(* Logix 5000 project; controller reports 1756-L63 rev 20.11; software revision 20.04; part 23 of 52 *)

        [1504].log_data[0].minminute := 40, [1504].log_data[0].maxminute := 40, [1504].log_data[0].valid := 1, [1504].log_data[1].valid := 1, [1504].log_data[2].valid := 1, [1504].log_data[3].valid := 1, [1504].log_data[4].valid := 1, [1504].log_data[5].valid := 1, [1504].log_data[6].valid := 1, [1504].log_data[7].valid := 1, [1504].log_data[8].valid := 1, [1504].log_data[9].valid := 1, [1504].log_data[10].valid := 1, [1504].log_data[11].valid := 1, [1504].log_data[12].valid := 1, [1504].log_data[13].valid := 1, [1504].log_data[14].valid := 1, [1504].log_data[15].valid := 1, [1504].log_data[16].valid := 1, [1504].log_data[17].valid := 1, [1504].log_data[18].valid := 1, [1504].log_data[19].valid := 1, [1504].time.Year := 2023, [1504].time.Month := 1, [1504].time.Day := 14, [1504].time.Hour := 21, [1504].time.Minute := 44, [1504].time.Second := 59, [1505].log_data[0].min := 1.0, [1505].log_data[0].max := 1.0, [1505].log_data[0].total := 300.0, [1505].log_data[0].time := 300.0, [1505].log_data[0].minminute := 45, [1505].log_data[0].maxminute := 45, [1505].log_data[0].valid := 1, [1505].log_data[1].valid := 1, [1505].log_data[2].valid := 1, [1505].log_data[3].valid := 1, [1505].log_data[4].valid := 1, [1505].log_data[5].valid := 1, [1505].log_data[6].valid := 1, [1505].log_data[7].valid := 1, [1505].log_data[8].valid := 1, [1505].log_data[9].valid := 1, [1505].log_data[10].valid := 1, [1505].log_data[11].valid := 1, [1505].log_data[12].valid := 1, [1505].log_data[13].valid := 1, [1505].log_data[14].valid := 1, [1505].log_data[15].valid := 1, [1505].log_data[16].valid := 1, [1505].log_data[17].valid := 1, [1505].log_data[18].valid := 1, [1505].log_data[19].valid := 1, [1505].time.Year := 2023, [1505].time.Month := 1, [1505].time.Day := 14, [1505].time.Hour := 21, [1505].time.Minute := 49, [1505].time.Second := 59,
        [1506].log_data[0].min := 1.0, [1506].log_data[0].max := 1.0, [1506].log_data[0].total := 300.0, [1506].log_data[0].time := 300.0, [1506].log_data[0].minminute := 50, [1506].log_data[0].maxminute := 50, [1506].log_data[0].valid := 1, [1506].log_data[1].valid := 1, [1506].log_data[2].valid := 1, [1506].log_data[3].valid := 1, [1506].log_data[4].valid := 1, [1506].log_data[5].valid := 1, [1506].log_data[6].valid := 1, [1506].log_data[7].valid := 1, [1506].log_data[8].valid := 1, [1506].log_data[9].valid := 1, [1506].log_data[10].valid := 1, [1506].log_data[11].valid := 1, [1506].log_data[12].valid := 1, [1506].log_data[13].valid := 1, [1506].log_data[14].valid := 1, [1506].log_data[15].valid := 1, [1506].log_data[16].valid := 1, [1506].log_data[17].valid := 1, [1506].log_data[18].valid := 1, [1506].log_data[19].valid := 1, [1506].time.Year := 2023, [1506].time.Month := 1, [1506].time.Day := 14, [1506].time.Hour := 21, [1506].time.Minute := 54, [1506].time.Second := 59, [1507].log_data[0].min := 1.0, [1507].log_data[0].max := 1.0, [1507].log_data[0].total := 300.0, [1507].log_data[0].time := 300.0, [1507].log_data[0].minminute := 55, [1507].log_data[0].maxminute := 55, [1507].log_data[0].valid := 1, [1507].log_data[1].valid := 1, [1507].log_data[2].valid := 1, [1507].log_data[3].valid := 1, [1507].log_data[4].valid := 1, [1507].log_data[5].valid := 1, [1507].log_data[6].valid := 1, [1507].log_data[7].valid := 1, [1507].log_data[8].valid := 1, [1507].log_data[9].valid := 1, [1507].log_data[10].valid := 1, [1507].log_data[11].valid := 1, [1507].log_data[12].valid := 1, [1507].log_data[13].valid := 1, [1507].log_data[14].valid := 1, [1507].log_data[15].valid := 1, [1507].log_data[16].valid := 1, [1507].log_data[17].valid := 1, [1507].log_data[18].valid := 1, [1507].log_data[19].valid := 1, [1507].time.Year := 2023, [1507].time.Month := 1,
        [1507].time.Day := 14, [1507].time.Hour := 21, [1507].time.Minute := 59, [1507].time.Second := 59, [1508].log_data[0].min := 1.0, [1508].log_data[0].max := 1.0, [1508].log_data[0].total := 300.0, [1508].log_data[0].time := 300.0, [1508].log_data[0].valid := 1, [1508].log_data[1].valid := 1, [1508].log_data[2].valid := 1, [1508].log_data[3].valid := 1, [1508].log_data[4].valid := 1, [1508].log_data[5].valid := 1, [1508].log_data[6].valid := 1, [1508].log_data[7].valid := 1, [1508].log_data[8].valid := 1, [1508].log_data[9].valid := 1, [1508].log_data[10].valid := 1, [1508].log_data[11].valid := 1, [1508].log_data[12].valid := 1, [1508].log_data[13].valid := 1, [1508].log_data[14].valid := 1, [1508].log_data[15].valid := 1, [1508].log_data[16].valid := 1, [1508].log_data[17].valid := 1, [1508].log_data[18].valid := 1, [1508].log_data[19].valid := 1, [1508].time.Year := 2023, [1508].time.Month := 1, [1508].time.Day := 14, [1508].time.Hour := 22, [1508].time.Minute := 4, [1508].time.Second := 59, [1509].log_data[0].min := 1.0, [1509].log_data[0].max := 1.0, [1509].log_data[0].total := 300.0, [1509].log_data[0].time := 300.0, [1509].log_data[0].minminute := 5, [1509].log_data[0].maxminute := 5, [1509].log_data[0].valid := 1, [1509].log_data[1].valid := 1, [1509].log_data[2].valid := 1, [1509].log_data[3].valid := 1, [1509].log_data[4].valid := 1, [1509].log_data[5].valid := 1, [1509].log_data[6].valid := 1, [1509].log_data[7].valid := 1, [1509].log_data[8].valid := 1, [1509].log_data[9].valid := 1, [1509].log_data[10].valid := 1, [1509].log_data[11].valid := 1, [1509].log_data[12].valid := 1, [1509].log_data[13].valid := 1, [1509].log_data[14].valid := 1, [1509].log_data[15].valid := 1, [1509].log_data[16].valid := 1, [1509].log_data[17].valid := 1, [1509].log_data[18].valid := 1, [1509].log_data[19].valid := 1,
        [1509].time.Year := 2023, [1509].time.Month := 1, [1509].time.Day := 14, [1509].time.Hour := 22, [1509].time.Minute := 9, [1509].time.Second := 59, [1510].log_data[0].min := 1.0, [1510].log_data[0].max := 1.0, [1510].log_data[0].total := 300.0, [1510].log_data[0].time := 300.0, [1510].log_data[0].minminute := 10, [1510].log_data[0].maxminute := 10, [1510].log_data[0].valid := 1, [1510].log_data[1].valid := 1, [1510].log_data[2].valid := 1, [1510].log_data[3].valid := 1, [1510].log_data[4].valid := 1, [1510].log_data[5].valid := 1, [1510].log_data[6].valid := 1, [1510].log_data[7].valid := 1, [1510].log_data[8].valid := 1, [1510].log_data[9].valid := 1, [1510].log_data[10].valid := 1, [1510].log_data[11].valid := 1, [1510].log_data[12].valid := 1, [1510].log_data[13].valid := 1, [1510].log_data[14].valid := 1, [1510].log_data[15].valid := 1, [1510].log_data[16].valid := 1, [1510].log_data[17].valid := 1, [1510].log_data[18].valid := 1, [1510].log_data[19].valid := 1, [1510].time.Year := 2023, [1510].time.Month := 1, [1510].time.Day := 14, [1510].time.Hour := 22, [1510].time.Minute := 14, [1510].time.Second := 59, [1511].log_data[0].min := 1.0, [1511].log_data[0].max := 1.0, [1511].log_data[0].total := 300.0, [1511].log_data[0].time := 300.0, [1511].log_data[0].minminute := 15, [1511].log_data[0].maxminute := 15, [1511].log_data[0].valid := 1, [1511].log_data[1].valid := 1, [1511].log_data[2].valid := 1, [1511].log_data[3].valid := 1, [1511].log_data[4].valid := 1, [1511].log_data[5].valid := 1, [1511].log_data[6].valid := 1, [1511].log_data[7].valid := 1, [1511].log_data[8].valid := 1, [1511].log_data[9].valid := 1, [1511].log_data[10].valid := 1, [1511].log_data[11].valid := 1, [1511].log_data[12].valid := 1, [1511].log_data[13].valid := 1, [1511].log_data[14].valid := 1, [1511].log_data[15].valid := 1,
        [1511].log_data[16].valid := 1, [1511].log_data[17].valid := 1, [1511].log_data[18].valid := 1, [1511].log_data[19].valid := 1, [1511].time.Year := 2023, [1511].time.Month := 1, [1511].time.Day := 14, [1511].time.Hour := 22, [1511].time.Minute := 19, [1511].time.Second := 59, [1512].log_data[0].min := 1.0, [1512].log_data[0].max := 1.0, [1512].log_data[0].total := 300.0, [1512].log_data[0].time := 300.0, [1512].log_data[0].minminute := 20, [1512].log_data[0].maxminute := 20, [1512].log_data[0].valid := 1, [1512].log_data[1].valid := 1, [1512].log_data[2].valid := 1, [1512].log_data[3].valid := 1, [1512].log_data[4].valid := 1, [1512].log_data[5].valid := 1, [1512].log_data[6].valid := 1, [1512].log_data[7].valid := 1, [1512].log_data[8].valid := 1, [1512].log_data[9].valid := 1, [1512].log_data[10].valid := 1, [1512].log_data[11].valid := 1, [1512].log_data[12].valid := 1, [1512].log_data[13].valid := 1, [1512].log_data[14].valid := 1, [1512].log_data[15].valid := 1, [1512].log_data[16].valid := 1, [1512].log_data[17].valid := 1, [1512].log_data[18].valid := 1, [1512].log_data[19].valid := 1, [1512].time.Year := 2023, [1512].time.Month := 1, [1512].time.Day := 14, [1512].time.Hour := 22, [1512].time.Minute := 24, [1512].time.Second := 59, [1513].log_data[0].min := 1.0, [1513].log_data[0].max := 1.0, [1513].log_data[0].total := 300.0, [1513].log_data[0].time := 300.0, [1513].log_data[0].minminute := 25, [1513].log_data[0].maxminute := 25, [1513].log_data[0].valid := 1, [1513].log_data[1].valid := 1, [1513].log_data[2].valid := 1, [1513].log_data[3].valid := 1, [1513].log_data[4].valid := 1, [1513].log_data[5].valid := 1, [1513].log_data[6].valid := 1, [1513].log_data[7].valid := 1, [1513].log_data[8].valid := 1, [1513].log_data[9].valid := 1, [1513].log_data[10].valid := 1, [1513].log_data[11].valid := 1,
        [1513].log_data[12].valid := 1, [1513].log_data[13].valid := 1, [1513].log_data[14].valid := 1, [1513].log_data[15].valid := 1, [1513].log_data[16].valid := 1, [1513].log_data[17].valid := 1, [1513].log_data[18].valid := 1, [1513].log_data[19].valid := 1, [1513].time.Year := 2023, [1513].time.Month := 1, [1513].time.Day := 14, [1513].time.Hour := 22, [1513].time.Minute := 29, [1513].time.Second := 59, [1514].log_data[0].min := 1.0, [1514].log_data[0].max := 1.0, [1514].log_data[0].total := 300.0, [1514].log_data[0].time := 300.0, [1514].log_data[0].minminute := 30, [1514].log_data[0].maxminute := 30, [1514].log_data[0].valid := 1, [1514].log_data[1].valid := 1, [1514].log_data[2].valid := 1, [1514].log_data[3].valid := 1, [1514].log_data[4].valid := 1, [1514].log_data[5].valid := 1, [1514].log_data[6].valid := 1, [1514].log_data[7].valid := 1, [1514].log_data[8].valid := 1, [1514].log_data[9].valid := 1, [1514].log_data[10].valid := 1, [1514].log_data[11].valid := 1, [1514].log_data[12].valid := 1, [1514].log_data[13].valid := 1, [1514].log_data[14].valid := 1, [1514].log_data[15].valid := 1, [1514].log_data[16].valid := 1, [1514].log_data[17].valid := 1, [1514].log_data[18].valid := 1, [1514].log_data[19].valid := 1, [1514].time.Year := 2023, [1514].time.Month := 1, [1514].time.Day := 14, [1514].time.Hour := 22, [1514].time.Minute := 34, [1514].time.Second := 59, [1515].log_data[0].min := 1.0, [1515].log_data[0].max := 1.0, [1515].log_data[0].total := 300.0, [1515].log_data[0].time := 300.0, [1515].log_data[0].minminute := 35, [1515].log_data[0].maxminute := 35, [1515].log_data[0].valid := 1, [1515].log_data[1].valid := 1, [1515].log_data[2].valid := 1, [1515].log_data[3].valid := 1, [1515].log_data[4].valid := 1, [1515].log_data[5].valid := 1, [1515].log_data[6].valid := 1, [1515].log_data[7].valid := 1,
        [1515].log_data[8].valid := 1, [1515].log_data[9].valid := 1, [1515].log_data[10].valid := 1, [1515].log_data[11].valid := 1, [1515].log_data[12].valid := 1, [1515].log_data[13].valid := 1, [1515].log_data[14].valid := 1, [1515].log_data[15].valid := 1, [1515].log_data[16].valid := 1, [1515].log_data[17].valid := 1, [1515].log_data[18].valid := 1, [1515].log_data[19].valid := 1, [1515].time.Year := 2023, [1515].time.Month := 1, [1515].time.Day := 14, [1515].time.Hour := 22, [1515].time.Minute := 39, [1515].time.Second := 59, [1516].log_data[0].min := 1.0, [1516].log_data[0].max := 1.0, [1516].log_data[0].total := 300.0, [1516].log_data[0].time := 300.0, [1516].log_data[0].minminute := 40, [1516].log_data[0].maxminute := 40, [1516].log_data[0].valid := 1, [1516].log_data[1].valid := 1, [1516].log_data[2].valid := 1, [1516].log_data[3].valid := 1, [1516].log_data[4].valid := 1, [1516].log_data[5].valid := 1, [1516].log_data[6].valid := 1, [1516].log_data[7].valid := 1, [1516].log_data[8].valid := 1, [1516].log_data[9].valid := 1, [1516].log_data[10].valid := 1, [1516].log_data[11].valid := 1, [1516].log_data[12].valid := 1, [1516].log_data[13].valid := 1, [1516].log_data[14].valid := 1, [1516].log_data[15].valid := 1, [1516].log_data[16].valid := 1, [1516].log_data[17].valid := 1, [1516].log_data[18].valid := 1, [1516].log_data[19].valid := 1, [1516].time.Year := 2023, [1516].time.Month := 1, [1516].time.Day := 14, [1516].time.Hour := 22, [1516].time.Minute := 44, [1516].time.Second := 59, [1517].log_data[0].min := 1.0, [1517].log_data[0].max := 1.0, [1517].log_data[0].total := 300.0, [1517].log_data[0].time := 300.0, [1517].log_data[0].minminute := 45, [1517].log_data[0].maxminute := 45, [1517].log_data[0].valid := 1, [1517].log_data[1].valid := 1, [1517].log_data[2].valid := 1, [1517].log_data[3].valid := 1,
        [1517].log_data[4].valid := 1, [1517].log_data[5].valid := 1, [1517].log_data[6].valid := 1, [1517].log_data[7].valid := 1, [1517].log_data[8].valid := 1, [1517].log_data[9].valid := 1, [1517].log_data[10].valid := 1, [1517].log_data[11].valid := 1, [1517].log_data[12].valid := 1, [1517].log_data[13].valid := 1, [1517].log_data[14].valid := 1, [1517].log_data[15].valid := 1, [1517].log_data[16].valid := 1, [1517].log_data[17].valid := 1, [1517].log_data[18].valid := 1, [1517].log_data[19].valid := 1, [1517].time.Year := 2023, [1517].time.Month := 1, [1517].time.Day := 14, [1517].time.Hour := 22, [1517].time.Minute := 49, [1517].time.Second := 59, [1518].log_data[0].min := 1.0, [1518].log_data[0].max := 1.0, [1518].log_data[0].total := 300.0, [1518].log_data[0].time := 300.0, [1518].log_data[0].minminute := 50, [1518].log_data[0].maxminute := 50, [1518].log_data[0].valid := 1, [1518].log_data[1].valid := 1, [1518].log_data[2].valid := 1, [1518].log_data[3].valid := 1, [1518].log_data[4].valid := 1, [1518].log_data[5].valid := 1, [1518].log_data[6].valid := 1, [1518].log_data[7].valid := 1, [1518].log_data[8].valid := 1, [1518].log_data[9].valid := 1, [1518].log_data[10].valid := 1, [1518].log_data[11].valid := 1, [1518].log_data[12].valid := 1, [1518].log_data[13].valid := 1, [1518].log_data[14].valid := 1, [1518].log_data[15].valid := 1, [1518].log_data[16].valid := 1, [1518].log_data[17].valid := 1, [1518].log_data[18].valid := 1, [1518].log_data[19].valid := 1, [1518].time.Year := 2023, [1518].time.Month := 1, [1518].time.Day := 14, [1518].time.Hour := 22, [1518].time.Minute := 54, [1518].time.Second := 59, [1519].log_data[0].min := 1.0, [1519].log_data[0].max := 1.0, [1519].log_data[0].total := 300.0, [1519].log_data[0].time := 300.0, [1519].log_data[0].minminute := 55, [1519].log_data[0].maxminute := 55,
        [1519].log_data[0].valid := 1, [1519].log_data[1].valid := 1, [1519].log_data[2].valid := 1, [1519].log_data[3].valid := 1, [1519].log_data[4].valid := 1, [1519].log_data[5].valid := 1, [1519].log_data[6].valid := 1, [1519].log_data[7].valid := 1, [1519].log_data[8].valid := 1, [1519].log_data[9].valid := 1, [1519].log_data[10].valid := 1, [1519].log_data[11].valid := 1, [1519].log_data[12].valid := 1, [1519].log_data[13].valid := 1, [1519].log_data[14].valid := 1, [1519].log_data[15].valid := 1, [1519].log_data[16].valid := 1, [1519].log_data[17].valid := 1, [1519].log_data[18].valid := 1, [1519].log_data[19].valid := 1, [1519].time.Year := 2023, [1519].time.Month := 1, [1519].time.Day := 14, [1519].time.Hour := 22, [1519].time.Minute := 59, [1519].time.Second := 59, [1520].log_data[0].min := 1.0, [1520].log_data[0].max := 1.0, [1520].log_data[0].total := 299.5, [1520].log_data[0].time := 299.5, [1520].log_data[0].valid := 1, [1520].log_data[1].valid := 1, [1520].log_data[2].valid := 1, [1520].log_data[3].valid := 1, [1520].log_data[4].valid := 1, [1520].log_data[5].valid := 1, [1520].log_data[6].valid := 1, [1520].log_data[7].valid := 1, [1520].log_data[8].valid := 1, [1520].log_data[9].valid := 1, [1520].log_data[10].valid := 1, [1520].log_data[11].valid := 1, [1520].log_data[12].valid := 1, [1520].log_data[13].valid := 1, [1520].log_data[14].valid := 1, [1520].log_data[15].valid := 1, [1520].log_data[16].valid := 1, [1520].log_data[17].valid := 1, [1520].log_data[18].valid := 1, [1520].log_data[19].valid := 1, [1520].time.Year := 2023, [1520].time.Month := 1, [1520].time.Day := 14, [1520].time.Hour := 23, [1520].time.Minute := 4, [1520].time.Second := 59, [1521].log_data[0].min := 1.0, [1521].log_data[0].max := 1.0, [1521].log_data[0].total := 300.0, [1521].log_data[0].time := 300.0,
        [1521].log_data[0].minminute := 5, [1521].log_data[0].maxminute := 5, [1521].log_data[0].valid := 1, [1521].log_data[1].valid := 1, [1521].log_data[2].valid := 1, [1521].log_data[3].valid := 1, [1521].log_data[4].valid := 1, [1521].log_data[5].valid := 1, [1521].log_data[6].valid := 1, [1521].log_data[7].valid := 1, [1521].log_data[8].valid := 1, [1521].log_data[9].valid := 1, [1521].log_data[10].valid := 1, [1521].log_data[11].valid := 1, [1521].log_data[12].valid := 1, [1521].log_data[13].valid := 1, [1521].log_data[14].valid := 1, [1521].log_data[15].valid := 1, [1521].log_data[16].valid := 1, [1521].log_data[17].valid := 1, [1521].log_data[18].valid := 1, [1521].log_data[19].valid := 1, [1521].time.Year := 2023, [1521].time.Month := 1, [1521].time.Day := 14, [1521].time.Hour := 23, [1521].time.Minute := 9, [1521].time.Second := 59, [1522].log_data[0].min := 1.0, [1522].log_data[0].max := 1.0, [1522].log_data[0].total := 300.0, [1522].log_data[0].time := 300.0, [1522].log_data[0].minminute := 10, [1522].log_data[0].maxminute := 10, [1522].log_data[0].valid := 1, [1522].log_data[1].valid := 1, [1522].log_data[2].valid := 1, [1522].log_data[3].valid := 1, [1522].log_data[4].valid := 1, [1522].log_data[5].valid := 1, [1522].log_data[6].valid := 1, [1522].log_data[7].valid := 1, [1522].log_data[8].valid := 1, [1522].log_data[9].valid := 1, [1522].log_data[10].valid := 1, [1522].log_data[11].valid := 1, [1522].log_data[12].valid := 1, [1522].log_data[13].valid := 1, [1522].log_data[14].valid := 1, [1522].log_data[15].valid := 1, [1522].log_data[16].valid := 1, [1522].log_data[17].valid := 1, [1522].log_data[18].valid := 1, [1522].log_data[19].valid := 1, [1522].time.Year := 2023, [1522].time.Month := 1, [1522].time.Day := 14, [1522].time.Hour := 23, [1522].time.Minute := 14, [1522].time.Second := 59,
        [1523].log_data[0].min := 1.0, [1523].log_data[0].max := 1.0, [1523].log_data[0].total := 300.0, [1523].log_data[0].time := 300.0, [1523].log_data[0].minminute := 15, [1523].log_data[0].maxminute := 15, [1523].log_data[0].valid := 1, [1523].log_data[1].valid := 1, [1523].log_data[2].valid := 1, [1523].log_data[3].valid := 1, [1523].log_data[4].valid := 1, [1523].log_data[5].valid := 1, [1523].log_data[6].valid := 1, [1523].log_data[7].valid := 1, [1523].log_data[8].valid := 1, [1523].log_data[9].valid := 1, [1523].log_data[10].valid := 1, [1523].log_data[11].valid := 1, [1523].log_data[12].valid := 1, [1523].log_data[13].valid := 1, [1523].log_data[14].valid := 1, [1523].log_data[15].valid := 1, [1523].log_data[16].valid := 1, [1523].log_data[17].valid := 1, [1523].log_data[18].valid := 1, [1523].log_data[19].valid := 1, [1523].time.Year := 2023, [1523].time.Month := 1, [1523].time.Day := 14, [1523].time.Hour := 23, [1523].time.Minute := 19, [1523].time.Second := 59, [1524].log_data[0].min := 1.0, [1524].log_data[0].max := 1.0, [1524].log_data[0].total := 300.0, [1524].log_data[0].time := 300.0, [1524].log_data[0].minminute := 20, [1524].log_data[0].maxminute := 20, [1524].log_data[0].valid := 1, [1524].log_data[1].valid := 1, [1524].log_data[2].valid := 1, [1524].log_data[3].valid := 1, [1524].log_data[4].valid := 1, [1524].log_data[5].valid := 1, [1524].log_data[6].valid := 1, [1524].log_data[7].valid := 1, [1524].log_data[8].valid := 1, [1524].log_data[9].valid := 1, [1524].log_data[10].valid := 1, [1524].log_data[11].valid := 1, [1524].log_data[12].valid := 1, [1524].log_data[13].valid := 1, [1524].log_data[14].valid := 1, [1524].log_data[15].valid := 1, [1524].log_data[16].valid := 1, [1524].log_data[17].valid := 1, [1524].log_data[18].valid := 1, [1524].log_data[19].valid := 1, [1524].time.Year := 2023, [1524].time.Month := 1,
        [1524].time.Day := 14, [1524].time.Hour := 23, [1524].time.Minute := 24, [1524].time.Second := 59, [1525].log_data[0].min := 1.0, [1525].log_data[0].max := 1.0, [1525].log_data[0].total := 300.0, [1525].log_data[0].time := 300.0, [1525].log_data[0].minminute := 25, [1525].log_data[0].maxminute := 25, [1525].log_data[0].valid := 1, [1525].log_data[1].valid := 1, [1525].log_data[2].valid := 1, [1525].log_data[3].valid := 1, [1525].log_data[4].valid := 1, [1525].log_data[5].valid := 1, [1525].log_data[6].valid := 1, [1525].log_data[7].valid := 1, [1525].log_data[8].valid := 1, [1525].log_data[9].valid := 1, [1525].log_data[10].valid := 1, [1525].log_data[11].valid := 1, [1525].log_data[12].valid := 1, [1525].log_data[13].valid := 1, [1525].log_data[14].valid := 1, [1525].log_data[15].valid := 1, [1525].log_data[16].valid := 1, [1525].log_data[17].valid := 1, [1525].log_data[18].valid := 1, [1525].log_data[19].valid := 1, [1525].time.Year := 2023, [1525].time.Month := 1, [1525].time.Day := 14, [1525].time.Hour := 23, [1525].time.Minute := 29, [1525].time.Second := 59, [1526].log_data[0].min := 1.0, [1526].log_data[0].max := 1.0, [1526].log_data[0].total := 300.0, [1526].log_data[0].time := 300.0, [1526].log_data[0].minminute := 30, [1526].log_data[0].maxminute := 30, [1526].log_data[0].valid := 1, [1526].log_data[1].valid := 1, [1526].log_data[2].valid := 1, [1526].log_data[3].valid := 1, [1526].log_data[4].valid := 1, [1526].log_data[5].valid := 1, [1526].log_data[6].valid := 1, [1526].log_data[7].valid := 1, [1526].log_data[8].valid := 1, [1526].log_data[9].valid := 1, [1526].log_data[10].valid := 1, [1526].log_data[11].valid := 1, [1526].log_data[12].valid := 1, [1526].log_data[13].valid := 1, [1526].log_data[14].valid := 1, [1526].log_data[15].valid := 1, [1526].log_data[16].valid := 1, [1526].log_data[17].valid := 1,
        [1526].log_data[18].valid := 1, [1526].log_data[19].valid := 1, [1526].time.Year := 2023, [1526].time.Month := 1, [1526].time.Day := 14, [1526].time.Hour := 23, [1526].time.Minute := 34, [1526].time.Second := 59, [1527].log_data[0].min := 1.0, [1527].log_data[0].max := 1.0, [1527].log_data[0].total := 300.0, [1527].log_data[0].time := 300.0, [1527].log_data[0].minminute := 35, [1527].log_data[0].maxminute := 35, [1527].log_data[0].valid := 1, [1527].log_data[1].valid := 1, [1527].log_data[2].valid := 1, [1527].log_data[3].valid := 1, [1527].log_data[4].valid := 1, [1527].log_data[5].valid := 1, [1527].log_data[6].valid := 1, [1527].log_data[7].valid := 1, [1527].log_data[8].valid := 1, [1527].log_data[9].valid := 1, [1527].log_data[10].valid := 1, [1527].log_data[11].valid := 1, [1527].log_data[12].valid := 1, [1527].log_data[13].valid := 1, [1527].log_data[14].valid := 1, [1527].log_data[15].valid := 1, [1527].log_data[16].valid := 1, [1527].log_data[17].valid := 1, [1527].log_data[18].valid := 1, [1527].log_data[19].valid := 1, [1527].time.Year := 2023, [1527].time.Month := 1, [1527].time.Day := 14, [1527].time.Hour := 23, [1527].time.Minute := 39, [1527].time.Second := 59, [1528].log_data[0].min := 1.0, [1528].log_data[0].max := 1.0, [1528].log_data[0].total := 300.0, [1528].log_data[0].time := 300.0, [1528].log_data[0].minminute := 40, [1528].log_data[0].maxminute := 40, [1528].log_data[0].valid := 1, [1528].log_data[1].valid := 1, [1528].log_data[2].valid := 1, [1528].log_data[3].valid := 1, [1528].log_data[4].valid := 1, [1528].log_data[5].valid := 1, [1528].log_data[6].valid := 1, [1528].log_data[7].valid := 1, [1528].log_data[8].valid := 1, [1528].log_data[9].valid := 1, [1528].log_data[10].valid := 1, [1528].log_data[11].valid := 1, [1528].log_data[12].valid := 1, [1528].log_data[13].valid := 1,
        [1528].log_data[14].valid := 1, [1528].log_data[15].valid := 1, [1528].log_data[16].valid := 1, [1528].log_data[17].valid := 1, [1528].log_data[18].valid := 1, [1528].log_data[19].valid := 1, [1528].time.Year := 2023, [1528].time.Month := 1, [1528].time.Day := 14, [1528].time.Hour := 23, [1528].time.Minute := 44, [1528].time.Second := 59, [1529].log_data[0].min := 1.0, [1529].log_data[0].max := 1.0, [1529].log_data[0].total := 300.0, [1529].log_data[0].time := 300.0, [1529].log_data[0].minminute := 45, [1529].log_data[0].maxminute := 45, [1529].log_data[0].valid := 1, [1529].log_data[1].valid := 1, [1529].log_data[2].valid := 1, [1529].log_data[3].valid := 1, [1529].log_data[4].valid := 1, [1529].log_data[5].valid := 1, [1529].log_data[6].valid := 1, [1529].log_data[7].valid := 1, [1529].log_data[8].valid := 1, [1529].log_data[9].valid := 1, [1529].log_data[10].valid := 1, [1529].log_data[11].valid := 1, [1529].log_data[12].valid := 1, [1529].log_data[13].valid := 1, [1529].log_data[14].valid := 1, [1529].log_data[15].valid := 1, [1529].log_data[16].valid := 1, [1529].log_data[17].valid := 1, [1529].log_data[18].valid := 1, [1529].log_data[19].valid := 1, [1529].time.Year := 2023, [1529].time.Month := 1, [1529].time.Day := 14, [1529].time.Hour := 23, [1529].time.Minute := 49, [1529].time.Second := 59, [1530].log_data[0].min := 1.0, [1530].log_data[0].max := 1.0, [1530].log_data[0].total := 300.0, [1530].log_data[0].time := 300.0, [1530].log_data[0].minminute := 50, [1530].log_data[0].maxminute := 50, [1530].log_data[0].valid := 1, [1530].log_data[1].valid := 1, [1530].log_data[2].valid := 1, [1530].log_data[3].valid := 1, [1530].log_data[4].valid := 1, [1530].log_data[5].valid := 1, [1530].log_data[6].valid := 1, [1530].log_data[7].valid := 1, [1530].log_data[8].valid := 1, [1530].log_data[9].valid := 1,
        [1530].log_data[10].valid := 1, [1530].log_data[11].valid := 1, [1530].log_data[12].valid := 1, [1530].log_data[13].valid := 1, [1530].log_data[14].valid := 1, [1530].log_data[15].valid := 1, [1530].log_data[16].valid := 1, [1530].log_data[17].valid := 1, [1530].log_data[18].valid := 1, [1530].log_data[19].valid := 1, [1530].time.Year := 2023, [1530].time.Month := 1, [1530].time.Day := 14, [1530].time.Hour := 23, [1530].time.Minute := 54, [1530].time.Second := 59, [1531].log_data[0].min := 1.0, [1531].log_data[0].max := 1.0, [1531].log_data[0].total := 300.0, [1531].log_data[0].time := 300.0, [1531].log_data[0].minminute := 55, [1531].log_data[0].maxminute := 55, [1531].log_data[0].valid := 1, [1531].log_data[1].valid := 1, [1531].log_data[2].valid := 1, [1531].log_data[3].valid := 1, [1531].log_data[4].valid := 1, [1531].log_data[5].valid := 1, [1531].log_data[6].valid := 1, [1531].log_data[7].valid := 1, [1531].log_data[8].valid := 1, [1531].log_data[9].valid := 1, [1531].log_data[10].valid := 1, [1531].log_data[11].valid := 1, [1531].log_data[12].valid := 1, [1531].log_data[13].valid := 1, [1531].log_data[14].valid := 1, [1531].log_data[15].valid := 1, [1531].log_data[16].valid := 1, [1531].log_data[17].valid := 1, [1531].log_data[18].valid := 1, [1531].log_data[19].valid := 1, [1531].time.Year := 2023, [1531].time.Month := 1, [1531].time.Day := 14, [1531].time.Hour := 23, [1531].time.Minute := 59, [1531].time.Second := 59, [1532].log_data[0].min := 1.0, [1532].log_data[0].max := 1.0, [1532].log_data[0].total := 300.0, [1532].log_data[0].time := 300.0, [1532].log_data[0].valid := 1, [1532].log_data[1].valid := 1, [1532].log_data[2].valid := 1, [1532].log_data[3].valid := 1, [1532].log_data[4].valid := 1, [1532].log_data[5].valid := 1, [1532].log_data[6].valid := 1, [1532].log_data[7].valid := 1,
        [1532].log_data[8].valid := 1, [1532].log_data[9].valid := 1, [1532].log_data[10].valid := 1, [1532].log_data[11].valid := 1, [1532].log_data[12].valid := 1, [1532].log_data[13].valid := 1, [1532].log_data[14].valid := 1, [1532].log_data[15].valid := 1, [1532].log_data[16].valid := 1, [1532].log_data[17].valid := 1, [1532].log_data[18].valid := 1, [1532].log_data[19].valid := 1, [1532].time.Year := 2023, [1532].time.Month := 1, [1532].time.Day := 15, [1532].time.Minute := 4, [1532].time.Second := 59, [1533].log_data[0].min := 1.0, [1533].log_data[0].max := 1.0, [1533].log_data[0].total := 300.0, [1533].log_data[0].time := 300.0, [1533].log_data[0].minminute := 5, [1533].log_data[0].maxminute := 5, [1533].log_data[0].valid := 1, [1533].log_data[1].valid := 1, [1533].log_data[2].valid := 1, [1533].log_data[3].valid := 1, [1533].log_data[4].valid := 1, [1533].log_data[5].valid := 1, [1533].log_data[6].valid := 1, [1533].log_data[7].valid := 1, [1533].log_data[8].valid := 1, [1533].log_data[9].valid := 1, [1533].log_data[10].valid := 1, [1533].log_data[11].valid := 1, [1533].log_data[12].valid := 1, [1533].log_data[13].valid := 1, [1533].log_data[14].valid := 1, [1533].log_data[15].valid := 1, [1533].log_data[16].valid := 1, [1533].log_data[17].valid := 1, [1533].log_data[18].valid := 1, [1533].log_data[19].valid := 1, [1533].time.Year := 2023, [1533].time.Month := 1, [1533].time.Day := 15, [1533].time.Minute := 9, [1533].time.Second := 59, [1534].log_data[0].min := 1.0, [1534].log_data[0].max := 1.0, [1534].log_data[0].total := 300.0, [1534].log_data[0].time := 300.0, [1534].log_data[0].minminute := 10, [1534].log_data[0].maxminute := 10, [1534].log_data[0].valid := 1, [1534].log_data[1].valid := 1, [1534].log_data[2].valid := 1, [1534].log_data[3].valid := 1, [1534].log_data[4].valid := 1, [1534].log_data[5].valid := 1,
        [1534].log_data[6].valid := 1, [1534].log_data[7].valid := 1, [1534].log_data[8].valid := 1, [1534].log_data[9].valid := 1, [1534].log_data[10].valid := 1, [1534].log_data[11].valid := 1, [1534].log_data[12].valid := 1, [1534].log_data[13].valid := 1, [1534].log_data[14].valid := 1, [1534].log_data[15].valid := 1, [1534].log_data[16].valid := 1, [1534].log_data[17].valid := 1, [1534].log_data[18].valid := 1, [1534].log_data[19].valid := 1, [1534].time.Year := 2023, [1534].time.Month := 1, [1534].time.Day := 15, [1534].time.Minute := 14, [1534].time.Second := 59, [1535].log_data[0].min := 1.0, [1535].log_data[0].max := 1.0, [1535].log_data[0].total := 300.0, [1535].log_data[0].time := 300.0, [1535].log_data[0].minminute := 15, [1535].log_data[0].maxminute := 15, [1535].log_data[0].valid := 1, [1535].log_data[1].valid := 1, [1535].log_data[2].valid := 1, [1535].log_data[3].valid := 1, [1535].log_data[4].valid := 1, [1535].log_data[5].valid := 1, [1535].log_data[6].valid := 1, [1535].log_data[7].valid := 1, [1535].log_data[8].valid := 1, [1535].log_data[9].valid := 1, [1535].log_data[10].valid := 1, [1535].log_data[11].valid := 1, [1535].log_data[12].valid := 1, [1535].log_data[13].valid := 1, [1535].log_data[14].valid := 1, [1535].log_data[15].valid := 1, [1535].log_data[16].valid := 1, [1535].log_data[17].valid := 1, [1535].log_data[18].valid := 1, [1535].log_data[19].valid := 1, [1535].time.Year := 2023, [1535].time.Month := 1, [1535].time.Day := 15, [1535].time.Minute := 19, [1535].time.Second := 59, [1536].log_data[0].min := 1.0, [1536].log_data[0].max := 1.0, [1536].log_data[0].total := 300.0, [1536].log_data[0].time := 300.0, [1536].log_data[0].minminute := 20, [1536].log_data[0].maxminute := 20, [1536].log_data[0].valid := 1, [1536].log_data[1].valid := 1, [1536].log_data[2].valid := 1, [1536].log_data[3].valid := 1,
        [1536].log_data[4].valid := 1, [1536].log_data[5].valid := 1, [1536].log_data[6].valid := 1, [1536].log_data[7].valid := 1, [1536].log_data[8].valid := 1, [1536].log_data[9].valid := 1, [1536].log_data[10].valid := 1, [1536].log_data[11].valid := 1, [1536].log_data[12].valid := 1, [1536].log_data[13].valid := 1, [1536].log_data[14].valid := 1, [1536].log_data[15].valid := 1, [1536].log_data[16].valid := 1, [1536].log_data[17].valid := 1, [1536].log_data[18].valid := 1, [1536].log_data[19].valid := 1, [1536].time.Year := 2023, [1536].time.Month := 1, [1536].time.Day := 15, [1536].time.Minute := 24, [1536].time.Second := 59, [1537].log_data[0].min := 1.0, [1537].log_data[0].max := 1.0, [1537].log_data[0].total := 300.0, [1537].log_data[0].time := 300.0, [1537].log_data[0].minminute := 25, [1537].log_data[0].maxminute := 25, [1537].log_data[0].valid := 1, [1537].log_data[1].valid := 1, [1537].log_data[2].valid := 1, [1537].log_data[3].valid := 1, [1537].log_data[4].valid := 1, [1537].log_data[5].valid := 1, [1537].log_data[6].valid := 1, [1537].log_data[7].valid := 1, [1537].log_data[8].valid := 1, [1537].log_data[9].valid := 1, [1537].log_data[10].valid := 1, [1537].log_data[11].valid := 1, [1537].log_data[12].valid := 1, [1537].log_data[13].valid := 1, [1537].log_data[14].valid := 1, [1537].log_data[15].valid := 1, [1537].log_data[16].valid := 1, [1537].log_data[17].valid := 1, [1537].log_data[18].valid := 1, [1537].log_data[19].valid := 1, [1537].time.Year := 2023, [1537].time.Month := 1, [1537].time.Day := 15, [1537].time.Minute := 29, [1537].time.Second := 59, [1538].log_data[0].min := 1.0, [1538].log_data[0].max := 1.0, [1538].log_data[0].total := 300.0, [1538].log_data[0].time := 300.0, [1538].log_data[0].minminute := 30, [1538].log_data[0].maxminute := 30, [1538].log_data[0].valid := 1, [1538].log_data[1].valid := 1,
        [1538].log_data[2].valid := 1, [1538].log_data[3].valid := 1, [1538].log_data[4].valid := 1, [1538].log_data[5].valid := 1, [1538].log_data[6].valid := 1, [1538].log_data[7].valid := 1, [1538].log_data[8].valid := 1, [1538].log_data[9].valid := 1, [1538].log_data[10].valid := 1, [1538].log_data[11].valid := 1, [1538].log_data[12].valid := 1, [1538].log_data[13].valid := 1, [1538].log_data[14].valid := 1, [1538].log_data[15].valid := 1, [1538].log_data[16].valid := 1, [1538].log_data[17].valid := 1, [1538].log_data[18].valid := 1, [1538].log_data[19].valid := 1, [1538].time.Year := 2023, [1538].time.Month := 1, [1538].time.Day := 15, [1538].time.Minute := 34, [1538].time.Second := 59, [1539].log_data[0].min := 1.0, [1539].log_data[0].max := 1.0, [1539].log_data[0].total := 300.0, [1539].log_data[0].time := 300.0, [1539].log_data[0].minminute := 35, [1539].log_data[0].maxminute := 35, [1539].log_data[0].valid := 1, [1539].log_data[1].valid := 1, [1539].log_data[2].valid := 1, [1539].log_data[3].valid := 1, [1539].log_data[4].valid := 1, [1539].log_data[5].valid := 1, [1539].log_data[6].valid := 1, [1539].log_data[7].valid := 1, [1539].log_data[8].valid := 1, [1539].log_data[9].valid := 1, [1539].log_data[10].valid := 1, [1539].log_data[11].valid := 1, [1539].log_data[12].valid := 1, [1539].log_data[13].valid := 1, [1539].log_data[14].valid := 1, [1539].log_data[15].valid := 1, [1539].log_data[16].valid := 1, [1539].log_data[17].valid := 1, [1539].log_data[18].valid := 1, [1539].log_data[19].valid := 1, [1539].time.Year := 2023, [1539].time.Month := 1, [1539].time.Day := 15, [1539].time.Minute := 39, [1539].time.Second := 59, [1540].log_data[0].min := 1.0, [1540].log_data[0].max := 1.0, [1540].log_data[0].total := 300.0, [1540].log_data[0].time := 300.0, [1540].log_data[0].minminute := 40, [1540].log_data[0].maxminute := 40,
        [1540].log_data[0].valid := 1, [1540].log_data[1].valid := 1, [1540].log_data[2].valid := 1, [1540].log_data[3].valid := 1, [1540].log_data[4].valid := 1, [1540].log_data[5].valid := 1, [1540].log_data[6].valid := 1, [1540].log_data[7].valid := 1, [1540].log_data[8].valid := 1, [1540].log_data[9].valid := 1, [1540].log_data[10].valid := 1, [1540].log_data[11].valid := 1, [1540].log_data[12].valid := 1, [1540].log_data[13].valid := 1, [1540].log_data[14].valid := 1, [1540].log_data[15].valid := 1, [1540].log_data[16].valid := 1, [1540].log_data[17].valid := 1, [1540].log_data[18].valid := 1, [1540].log_data[19].valid := 1, [1540].time.Year := 2023, [1540].time.Month := 1, [1540].time.Day := 15, [1540].time.Minute := 44, [1540].time.Second := 59, [1541].log_data[0].min := 1.0, [1541].log_data[0].max := 1.0, [1541].log_data[0].total := 300.0, [1541].log_data[0].time := 300.0, [1541].log_data[0].minminute := 45, [1541].log_data[0].maxminute := 45, [1541].log_data[0].valid := 1, [1541].log_data[1].valid := 1, [1541].log_data[2].valid := 1, [1541].log_data[3].valid := 1, [1541].log_data[4].valid := 1, [1541].log_data[5].valid := 1, [1541].log_data[6].valid := 1, [1541].log_data[7].valid := 1, [1541].log_data[8].valid := 1, [1541].log_data[9].valid := 1, [1541].log_data[10].valid := 1, [1541].log_data[11].valid := 1, [1541].log_data[12].valid := 1, [1541].log_data[13].valid := 1, [1541].log_data[14].valid := 1, [1541].log_data[15].valid := 1, [1541].log_data[16].valid := 1, [1541].log_data[17].valid := 1, [1541].log_data[18].valid := 1, [1541].log_data[19].valid := 1, [1541].time.Year := 2023, [1541].time.Month := 1, [1541].time.Day := 15, [1541].time.Minute := 49, [1541].time.Second := 59, [1542].log_data[0].min := 1.0, [1542].log_data[0].max := 1.0, [1542].log_data[0].total := 300.0, [1542].log_data[0].time := 300.0,
        [1542].log_data[0].minminute := 50, [1542].log_data[0].maxminute := 50, [1542].log_data[0].valid := 1, [1542].log_data[1].valid := 1, [1542].log_data[2].valid := 1, [1542].log_data[3].valid := 1, [1542].log_data[4].valid := 1, [1542].log_data[5].valid := 1, [1542].log_data[6].valid := 1, [1542].log_data[7].valid := 1, [1542].log_data[8].valid := 1, [1542].log_data[9].valid := 1, [1542].log_data[10].valid := 1, [1542].log_data[11].valid := 1, [1542].log_data[12].valid := 1, [1542].log_data[13].valid := 1, [1542].log_data[14].valid := 1, [1542].log_data[15].valid := 1, [1542].log_data[16].valid := 1, [1542].log_data[17].valid := 1, [1542].log_data[18].valid := 1, [1542].log_data[19].valid := 1, [1542].time.Year := 2023, [1542].time.Month := 1, [1542].time.Day := 15, [1542].time.Minute := 54, [1542].time.Second := 59, [1543].log_data[0].min := 1.0, [1543].log_data[0].max := 1.0, [1543].log_data[0].total := 300.0, [1543].log_data[0].time := 300.0, [1543].log_data[0].minminute := 55, [1543].log_data[0].maxminute := 55, [1543].log_data[0].valid := 1, [1543].log_data[1].valid := 1, [1543].log_data[2].valid := 1, [1543].log_data[3].valid := 1, [1543].log_data[4].valid := 1, [1543].log_data[5].valid := 1, [1543].log_data[6].valid := 1, [1543].log_data[7].valid := 1, [1543].log_data[8].valid := 1, [1543].log_data[9].valid := 1, [1543].log_data[10].valid := 1, [1543].log_data[11].valid := 1, [1543].log_data[12].valid := 1, [1543].log_data[13].valid := 1, [1543].log_data[14].valid := 1, [1543].log_data[15].valid := 1, [1543].log_data[16].valid := 1, [1543].log_data[17].valid := 1, [1543].log_data[18].valid := 1, [1543].log_data[19].valid := 1, [1543].time.Year := 2023, [1543].time.Month := 1, [1543].time.Day := 15, [1543].time.Minute := 59, [1543].time.Second := 59, [1544].log_data[0].min := 1.0, [1544].log_data[0].max := 1.0,
        [1544].log_data[0].total := 300.0, [1544].log_data[0].time := 300.0, [1544].log_data[0].valid := 1, [1544].log_data[1].valid := 1, [1544].log_data[2].valid := 1, [1544].log_data[3].valid := 1, [1544].log_data[4].valid := 1, [1544].log_data[5].valid := 1, [1544].log_data[6].valid := 1, [1544].log_data[7].valid := 1, [1544].log_data[8].valid := 1, [1544].log_data[9].valid := 1, [1544].log_data[10].valid := 1, [1544].log_data[11].valid := 1, [1544].log_data[12].valid := 1, [1544].log_data[13].valid := 1, [1544].log_data[14].valid := 1, [1544].log_data[15].valid := 1, [1544].log_data[16].valid := 1, [1544].log_data[17].valid := 1, [1544].log_data[18].valid := 1, [1544].log_data[19].valid := 1, [1544].time.Year := 2023, [1544].time.Month := 1, [1544].time.Day := 15, [1544].time.Hour := 1, [1544].time.Minute := 4, [1544].time.Second := 59, [1545].log_data[0].min := 1.0, [1545].log_data[0].max := 1.0, [1545].log_data[0].total := 300.0, [1545].log_data[0].time := 300.0, [1545].log_data[0].minminute := 5, [1545].log_data[0].maxminute := 5, [1545].log_data[0].valid := 1, [1545].log_data[1].valid := 1, [1545].log_data[2].valid := 1, [1545].log_data[3].valid := 1, [1545].log_data[4].valid := 1, [1545].log_data[5].valid := 1, [1545].log_data[6].valid := 1, [1545].log_data[7].valid := 1, [1545].log_data[8].valid := 1, [1545].log_data[9].valid := 1, [1545].log_data[10].valid := 1, [1545].log_data[11].valid := 1, [1545].log_data[12].valid := 1, [1545].log_data[13].valid := 1, [1545].log_data[14].valid := 1, [1545].log_data[15].valid := 1, [1545].log_data[16].valid := 1, [1545].log_data[17].valid := 1, [1545].log_data[18].valid := 1, [1545].log_data[19].valid := 1, [1545].time.Year := 2023, [1545].time.Month := 1, [1545].time.Day := 15, [1545].time.Hour := 1, [1545].time.Minute := 9, [1545].time.Second := 59,
        [1546].log_data[0].min := 1.0, [1546].log_data[0].max := 1.0, [1546].log_data[0].total := 300.0, [1546].log_data[0].time := 300.0, [1546].log_data[0].minminute := 10, [1546].log_data[0].maxminute := 10, [1546].log_data[0].valid := 1, [1546].log_data[1].valid := 1, [1546].log_data[2].valid := 1, [1546].log_data[3].valid := 1, [1546].log_data[4].valid := 1, [1546].log_data[5].valid := 1, [1546].log_data[6].valid := 1, [1546].log_data[7].valid := 1, [1546].log_data[8].valid := 1, [1546].log_data[9].valid := 1, [1546].log_data[10].valid := 1, [1546].log_data[11].valid := 1, [1546].log_data[12].valid := 1, [1546].log_data[13].valid := 1, [1546].log_data[14].valid := 1, [1546].log_data[15].valid := 1, [1546].log_data[16].valid := 1, [1546].log_data[17].valid := 1, [1546].log_data[18].valid := 1, [1546].log_data[19].valid := 1, [1546].time.Year := 2023, [1546].time.Month := 1, [1546].time.Day := 15, [1546].time.Hour := 1, [1546].time.Minute := 14, [1546].time.Second := 59, [1547].log_data[0].min := 1.0, [1547].log_data[0].max := 1.0, [1547].log_data[0].total := 300.0, [1547].log_data[0].time := 300.0, [1547].log_data[0].minminute := 15, [1547].log_data[0].maxminute := 15, [1547].log_data[0].valid := 1, [1547].log_data[1].valid := 1, [1547].log_data[2].valid := 1, [1547].log_data[3].valid := 1, [1547].log_data[4].valid := 1, [1547].log_data[5].valid := 1, [1547].log_data[6].valid := 1, [1547].log_data[7].valid := 1, [1547].log_data[8].valid := 1, [1547].log_data[9].valid := 1, [1547].log_data[10].valid := 1, [1547].log_data[11].valid := 1, [1547].log_data[12].valid := 1, [1547].log_data[13].valid := 1, [1547].log_data[14].valid := 1, [1547].log_data[15].valid := 1, [1547].log_data[16].valid := 1, [1547].log_data[17].valid := 1, [1547].log_data[18].valid := 1, [1547].log_data[19].valid := 1, [1547].time.Year := 2023, [1547].time.Month := 1,
        [1547].time.Day := 15, [1547].time.Hour := 1, [1547].time.Minute := 19, [1547].time.Second := 59, [1548].log_data[0].min := 1.0, [1548].log_data[0].max := 1.0, [1548].log_data[0].total := 300.0, [1548].log_data[0].time := 300.0, [1548].log_data[0].minminute := 20, [1548].log_data[0].maxminute := 20, [1548].log_data[0].valid := 1, [1548].log_data[1].valid := 1, [1548].log_data[2].valid := 1, [1548].log_data[3].valid := 1, [1548].log_data[4].valid := 1, [1548].log_data[5].valid := 1, [1548].log_data[6].valid := 1, [1548].log_data[7].valid := 1, [1548].log_data[8].valid := 1, [1548].log_data[9].valid := 1, [1548].log_data[10].valid := 1, [1548].log_data[11].valid := 1, [1548].log_data[12].valid := 1, [1548].log_data[13].valid := 1, [1548].log_data[14].valid := 1, [1548].log_data[15].valid := 1, [1548].log_data[16].valid := 1, [1548].log_data[17].valid := 1, [1548].log_data[18].valid := 1, [1548].log_data[19].valid := 1, [1548].time.Year := 2023, [1548].time.Month := 1, [1548].time.Day := 15, [1548].time.Hour := 1, [1548].time.Minute := 24, [1548].time.Second := 59, [1549].log_data[0].min := 1.0, [1549].log_data[0].max := 1.0, [1549].log_data[0].total := 300.0, [1549].log_data[0].time := 300.0, [1549].log_data[0].minminute := 25, [1549].log_data[0].maxminute := 25, [1549].log_data[0].valid := 1, [1549].log_data[1].valid := 1, [1549].log_data[2].valid := 1, [1549].log_data[3].valid := 1, [1549].log_data[4].valid := 1, [1549].log_data[5].valid := 1, [1549].log_data[6].valid := 1, [1549].log_data[7].valid := 1, [1549].log_data[8].valid := 1, [1549].log_data[9].valid := 1, [1549].log_data[10].valid := 1, [1549].log_data[11].valid := 1, [1549].log_data[12].valid := 1, [1549].log_data[13].valid := 1, [1549].log_data[14].valid := 1, [1549].log_data[15].valid := 1, [1549].log_data[16].valid := 1, [1549].log_data[17].valid := 1,
        [1549].log_data[18].valid := 1, [1549].log_data[19].valid := 1, [1549].time.Year := 2023, [1549].time.Month := 1, [1549].time.Day := 15, [1549].time.Hour := 1, [1549].time.Minute := 29, [1549].time.Second := 59, [1550].log_data[0].min := 1.0, [1550].log_data[0].max := 1.0, [1550].log_data[0].total := 300.0, [1550].log_data[0].time := 300.0, [1550].log_data[0].minminute := 30, [1550].log_data[0].maxminute := 30, [1550].log_data[0].valid := 1, [1550].log_data[1].valid := 1, [1550].log_data[2].valid := 1, [1550].log_data[3].valid := 1, [1550].log_data[4].valid := 1, [1550].log_data[5].valid := 1, [1550].log_data[6].valid := 1, [1550].log_data[7].valid := 1, [1550].log_data[8].valid := 1, [1550].log_data[9].valid := 1, [1550].log_data[10].valid := 1, [1550].log_data[11].valid := 1, [1550].log_data[12].valid := 1, [1550].log_data[13].valid := 1, [1550].log_data[14].valid := 1, [1550].log_data[15].valid := 1, [1550].log_data[16].valid := 1, [1550].log_data[17].valid := 1, [1550].log_data[18].valid := 1, [1550].log_data[19].valid := 1, [1550].time.Year := 2023, [1550].time.Month := 1, [1550].time.Day := 15, [1550].time.Hour := 1, [1550].time.Minute := 34, [1550].time.Second := 59, [1551].log_data[0].min := 1.0, [1551].log_data[0].max := 1.0, [1551].log_data[0].total := 300.0, [1551].log_data[0].time := 300.0, [1551].log_data[0].minminute := 35, [1551].log_data[0].maxminute := 35, [1551].log_data[0].valid := 1, [1551].log_data[1].valid := 1, [1551].log_data[2].valid := 1, [1551].log_data[3].valid := 1, [1551].log_data[4].valid := 1, [1551].log_data[5].valid := 1, [1551].log_data[6].valid := 1, [1551].log_data[7].valid := 1, [1551].log_data[8].valid := 1, [1551].log_data[9].valid := 1, [1551].log_data[10].valid := 1, [1551].log_data[11].valid := 1, [1551].log_data[12].valid := 1, [1551].log_data[13].valid := 1,
        [1551].log_data[14].valid := 1, [1551].log_data[15].valid := 1, [1551].log_data[16].valid := 1, [1551].log_data[17].valid := 1, [1551].log_data[18].valid := 1, [1551].log_data[19].valid := 1, [1551].time.Year := 2023, [1551].time.Month := 1, [1551].time.Day := 15, [1551].time.Hour := 1, [1551].time.Minute := 39, [1551].time.Second := 59, [1552].log_data[0].min := 1.0, [1552].log_data[0].max := 1.0, [1552].log_data[0].total := 300.0, [1552].log_data[0].time := 300.0, [1552].log_data[0].minminute := 40, [1552].log_data[0].maxminute := 40, [1552].log_data[0].valid := 1, [1552].log_data[1].valid := 1, [1552].log_data[2].valid := 1, [1552].log_data[3].valid := 1, [1552].log_data[4].valid := 1, [1552].log_data[5].valid := 1, [1552].log_data[6].valid := 1, [1552].log_data[7].valid := 1, [1552].log_data[8].valid := 1, [1552].log_data[9].valid := 1, [1552].log_data[10].valid := 1, [1552].log_data[11].valid := 1, [1552].log_data[12].valid := 1, [1552].log_data[13].valid := 1, [1552].log_data[14].valid := 1, [1552].log_data[15].valid := 1, [1552].log_data[16].valid := 1, [1552].log_data[17].valid := 1, [1552].log_data[18].valid := 1, [1552].log_data[19].valid := 1, [1552].time.Year := 2023, [1552].time.Month := 1, [1552].time.Day := 15, [1552].time.Hour := 1, [1552].time.Minute := 44, [1552].time.Second := 59, [1553].log_data[0].min := 1.0, [1553].log_data[0].max := 1.0, [1553].log_data[0].total := 300.0, [1553].log_data[0].time := 300.0, [1553].log_data[0].minminute := 45, [1553].log_data[0].maxminute := 45, [1553].log_data[0].valid := 1, [1553].log_data[1].valid := 1, [1553].log_data[2].valid := 1, [1553].log_data[3].valid := 1, [1553].log_data[4].valid := 1, [1553].log_data[5].valid := 1, [1553].log_data[6].valid := 1, [1553].log_data[7].valid := 1, [1553].log_data[8].valid := 1, [1553].log_data[9].valid := 1,
        [1553].log_data[10].valid := 1, [1553].log_data[11].valid := 1, [1553].log_data[12].valid := 1, [1553].log_data[13].valid := 1, [1553].log_data[14].valid := 1, [1553].log_data[15].valid := 1, [1553].log_data[16].valid := 1, [1553].log_data[17].valid := 1, [1553].log_data[18].valid := 1, [1553].log_data[19].valid := 1, [1553].time.Year := 2023, [1553].time.Month := 1, [1553].time.Day := 15, [1553].time.Hour := 1, [1553].time.Minute := 49, [1553].time.Second := 59, [1554].log_data[0].min := 1.0, [1554].log_data[0].max := 1.0, [1554].log_data[0].total := 300.0, [1554].log_data[0].time := 300.0, [1554].log_data[0].minminute := 50, [1554].log_data[0].maxminute := 50, [1554].log_data[0].valid := 1, [1554].log_data[1].valid := 1, [1554].log_data[2].valid := 1, [1554].log_data[3].valid := 1, [1554].log_data[4].valid := 1, [1554].log_data[5].valid := 1, [1554].log_data[6].valid := 1, [1554].log_data[7].valid := 1, [1554].log_data[8].valid := 1, [1554].log_data[9].valid := 1, [1554].log_data[10].valid := 1, [1554].log_data[11].valid := 1, [1554].log_data[12].valid := 1, [1554].log_data[13].valid := 1, [1554].log_data[14].valid := 1, [1554].log_data[15].valid := 1, [1554].log_data[16].valid := 1, [1554].log_data[17].valid := 1, [1554].log_data[18].valid := 1, [1554].log_data[19].valid := 1, [1554].time.Year := 2023, [1554].time.Month := 1, [1554].time.Day := 15, [1554].time.Hour := 1, [1554].time.Minute := 54, [1554].time.Second := 59, [1555].log_data[0].min := 1.0, [1555].log_data[0].max := 1.0, [1555].log_data[0].total := 300.0, [1555].log_data[0].time := 300.0, [1555].log_data[0].minminute := 55, [1555].log_data[0].maxminute := 55, [1555].log_data[0].valid := 1, [1555].log_data[1].valid := 1, [1555].log_data[2].valid := 1, [1555].log_data[3].valid := 1, [1555].log_data[4].valid := 1, [1555].log_data[5].valid := 1,
        [1555].log_data[6].valid := 1, [1555].log_data[7].valid := 1, [1555].log_data[8].valid := 1, [1555].log_data[9].valid := 1, [1555].log_data[10].valid := 1, [1555].log_data[11].valid := 1, [1555].log_data[12].valid := 1, [1555].log_data[13].valid := 1, [1555].log_data[14].valid := 1, [1555].log_data[15].valid := 1, [1555].log_data[16].valid := 1, [1555].log_data[17].valid := 1, [1555].log_data[18].valid := 1, [1555].log_data[19].valid := 1, [1555].time.Year := 2023, [1555].time.Month := 1, [1555].time.Day := 15, [1555].time.Hour := 1, [1555].time.Minute := 59, [1555].time.Second := 59, [1556].log_data[0].min := 1.0, [1556].log_data[0].max := 1.0, [1556].log_data[0].total := 300.0, [1556].log_data[0].time := 300.0, [1556].log_data[0].valid := 1, [1556].log_data[1].valid := 1, [1556].log_data[2].valid := 1, [1556].log_data[3].valid := 1, [1556].log_data[4].valid := 1, [1556].log_data[5].valid := 1, [1556].log_data[6].valid := 1, [1556].log_data[7].valid := 1, [1556].log_data[8].valid := 1, [1556].log_data[9].valid := 1, [1556].log_data[10].valid := 1, [1556].log_data[11].valid := 1, [1556].log_data[12].valid := 1, [1556].log_data[13].valid := 1, [1556].log_data[14].valid := 1, [1556].log_data[15].valid := 1, [1556].log_data[16].valid := 1, [1556].log_data[17].valid := 1, [1556].log_data[18].valid := 1, [1556].log_data[19].valid := 1, [1556].time.Year := 2023, [1556].time.Month := 1, [1556].time.Day := 15, [1556].time.Hour := 2, [1556].time.Minute := 4, [1556].time.Second := 59, [1557].log_data[0].min := 1.0, [1557].log_data[0].max := 1.0, [1557].log_data[0].total := 300.0, [1557].log_data[0].time := 300.0, [1557].log_data[0].minminute := 5, [1557].log_data[0].maxminute := 5, [1557].log_data[0].valid := 1, [1557].log_data[1].valid := 1, [1557].log_data[2].valid := 1, [1557].log_data[3].valid := 1,
        [1557].log_data[4].valid := 1, [1557].log_data[5].valid := 1, [1557].log_data[6].valid := 1, [1557].log_data[7].valid := 1, [1557].log_data[8].valid := 1, [1557].log_data[9].valid := 1, [1557].log_data[10].valid := 1, [1557].log_data[11].valid := 1, [1557].log_data[12].valid := 1, [1557].log_data[13].valid := 1, [1557].log_data[14].valid := 1, [1557].log_data[15].valid := 1, [1557].log_data[16].valid := 1, [1557].log_data[17].valid := 1, [1557].log_data[18].valid := 1, [1557].log_data[19].valid := 1, [1557].time.Year := 2023, [1557].time.Month := 1, [1557].time.Day := 15, [1557].time.Hour := 2, [1557].time.Minute := 9, [1557].time.Second := 59, [1558].log_data[0].min := 1.0, [1558].log_data[0].max := 1.0, [1558].log_data[0].total := 300.0, [1558].log_data[0].time := 300.0, [1558].log_data[0].minminute := 10, [1558].log_data[0].maxminute := 10, [1558].log_data[0].valid := 1, [1558].log_data[1].valid := 1, [1558].log_data[2].valid := 1, [1558].log_data[3].valid := 1, [1558].log_data[4].valid := 1, [1558].log_data[5].valid := 1, [1558].log_data[6].valid := 1, [1558].log_data[7].valid := 1, [1558].log_data[8].valid := 1, [1558].log_data[9].valid := 1, [1558].log_data[10].valid := 1, [1558].log_data[11].valid := 1, [1558].log_data[12].valid := 1, [1558].log_data[13].valid := 1, [1558].log_data[14].valid := 1, [1558].log_data[15].valid := 1, [1558].log_data[16].valid := 1, [1558].log_data[17].valid := 1, [1558].log_data[18].valid := 1, [1558].log_data[19].valid := 1, [1558].time.Year := 2023, [1558].time.Month := 1, [1558].time.Day := 15, [1558].time.Hour := 2, [1558].time.Minute := 14, [1558].time.Second := 59, [1559].log_data[0].min := 1.0, [1559].log_data[0].max := 1.0, [1559].log_data[0].total := 300.0, [1559].log_data[0].time := 300.0, [1559].log_data[0].minminute := 15, [1559].log_data[0].maxminute := 15,
        [1559].log_data[0].valid := 1, [1559].log_data[1].valid := 1, [1559].log_data[2].valid := 1, [1559].log_data[3].valid := 1, [1559].log_data[4].valid := 1, [1559].log_data[5].valid := 1, [1559].log_data[6].valid := 1, [1559].log_data[7].valid := 1, [1559].log_data[8].valid := 1, [1559].log_data[9].valid := 1, [1559].log_data[10].valid := 1, [1559].log_data[11].valid := 1, [1559].log_data[12].valid := 1, [1559].log_data[13].valid := 1, [1559].log_data[14].valid := 1, [1559].log_data[15].valid := 1, [1559].log_data[16].valid := 1, [1559].log_data[17].valid := 1, [1559].log_data[18].valid := 1, [1559].log_data[19].valid := 1, [1559].time.Year := 2023, [1559].time.Month := 1, [1559].time.Day := 15, [1559].time.Hour := 2, [1559].time.Minute := 19, [1559].time.Second := 59, [1560].log_data[0].min := 1.0, [1560].log_data[0].max := 1.0, [1560].log_data[0].total := 300.0, [1560].log_data[0].time := 300.0, [1560].log_data[0].minminute := 20, [1560].log_data[0].maxminute := 20, [1560].log_data[0].valid := 1, [1560].log_data[1].valid := 1, [1560].log_data[2].valid := 1, [1560].log_data[3].valid := 1, [1560].log_data[4].valid := 1, [1560].log_data[5].valid := 1, [1560].log_data[6].valid := 1, [1560].log_data[7].valid := 1, [1560].log_data[8].valid := 1, [1560].log_data[9].valid := 1, [1560].log_data[10].valid := 1, [1560].log_data[11].valid := 1, [1560].log_data[12].valid := 1, [1560].log_data[13].valid := 1, [1560].log_data[14].valid := 1, [1560].log_data[15].valid := 1, [1560].log_data[16].valid := 1, [1560].log_data[17].valid := 1, [1560].log_data[18].valid := 1, [1560].log_data[19].valid := 1, [1560].time.Year := 2023, [1560].time.Month := 1, [1560].time.Day := 15, [1560].time.Hour := 2, [1560].time.Minute := 24, [1560].time.Second := 59, [1561].log_data[0].min := 1.0, [1561].log_data[0].max := 1.0,
        [1561].log_data[0].total := 300.0, [1561].log_data[0].time := 300.0, [1561].log_data[0].minminute := 25, [1561].log_data[0].maxminute := 25, [1561].log_data[0].valid := 1, [1561].log_data[1].valid := 1, [1561].log_data[2].valid := 1, [1561].log_data[3].valid := 1, [1561].log_data[4].valid := 1, [1561].log_data[5].valid := 1, [1561].log_data[6].valid := 1, [1561].log_data[7].valid := 1, [1561].log_data[8].valid := 1, [1561].log_data[9].valid := 1, [1561].log_data[10].valid := 1, [1561].log_data[11].valid := 1, [1561].log_data[12].valid := 1, [1561].log_data[13].valid := 1, [1561].log_data[14].valid := 1, [1561].log_data[15].valid := 1, [1561].log_data[16].valid := 1, [1561].log_data[17].valid := 1, [1561].log_data[18].valid := 1, [1561].log_data[19].valid := 1, [1561].time.Year := 2023, [1561].time.Month := 1, [1561].time.Day := 15, [1561].time.Hour := 2, [1561].time.Minute := 29, [1561].time.Second := 59, [1562].log_data[0].min := 1.0, [1562].log_data[0].max := 1.0, [1562].log_data[0].total := 300.0, [1562].log_data[0].time := 300.0, [1562].log_data[0].minminute := 30, [1562].log_data[0].maxminute := 30, [1562].log_data[0].valid := 1, [1562].log_data[1].valid := 1, [1562].log_data[2].valid := 1, [1562].log_data[3].valid := 1, [1562].log_data[4].valid := 1, [1562].log_data[5].valid := 1, [1562].log_data[6].valid := 1, [1562].log_data[7].valid := 1, [1562].log_data[8].valid := 1, [1562].log_data[9].valid := 1, [1562].log_data[10].valid := 1, [1562].log_data[11].valid := 1, [1562].log_data[12].valid := 1, [1562].log_data[13].valid := 1, [1562].log_data[14].valid := 1, [1562].log_data[15].valid := 1, [1562].log_data[16].valid := 1, [1562].log_data[17].valid := 1, [1562].log_data[18].valid := 1, [1562].log_data[19].valid := 1, [1562].time.Year := 2023, [1562].time.Month := 1, [1562].time.Day := 15, [1562].time.Hour := 2,
        [1562].time.Minute := 34, [1562].time.Second := 59, [1563].log_data[0].min := 1.0, [1563].log_data[0].max := 1.0, [1563].log_data[0].total := 300.0, [1563].log_data[0].time := 300.0, [1563].log_data[0].minminute := 35, [1563].log_data[0].maxminute := 35, [1563].log_data[0].valid := 1, [1563].log_data[1].valid := 1, [1563].log_data[2].valid := 1, [1563].log_data[3].valid := 1, [1563].log_data[4].valid := 1, [1563].log_data[5].valid := 1, [1563].log_data[6].valid := 1, [1563].log_data[7].valid := 1, [1563].log_data[8].valid := 1, [1563].log_data[9].valid := 1, [1563].log_data[10].valid := 1, [1563].log_data[11].valid := 1, [1563].log_data[12].valid := 1, [1563].log_data[13].valid := 1, [1563].log_data[14].valid := 1, [1563].log_data[15].valid := 1, [1563].log_data[16].valid := 1, [1563].log_data[17].valid := 1, [1563].log_data[18].valid := 1, [1563].log_data[19].valid := 1, [1563].time.Year := 2023, [1563].time.Month := 1, [1563].time.Day := 15, [1563].time.Hour := 2, [1563].time.Minute := 39, [1563].time.Second := 59, [1564].log_data[0].min := 1.0, [1564].log_data[0].max := 1.0, [1564].log_data[0].total := 300.0, [1564].log_data[0].time := 300.0, [1564].log_data[0].minminute := 40, [1564].log_data[0].maxminute := 40, [1564].log_data[0].valid := 1, [1564].log_data[1].valid := 1, [1564].log_data[2].valid := 1, [1564].log_data[3].valid := 1, [1564].log_data[4].valid := 1, [1564].log_data[5].valid := 1, [1564].log_data[6].valid := 1, [1564].log_data[7].valid := 1, [1564].log_data[8].valid := 1, [1564].log_data[9].valid := 1, [1564].log_data[10].valid := 1, [1564].log_data[11].valid := 1, [1564].log_data[12].valid := 1, [1564].log_data[13].valid := 1, [1564].log_data[14].valid := 1, [1564].log_data[15].valid := 1, [1564].log_data[16].valid := 1, [1564].log_data[17].valid := 1, [1564].log_data[18].valid := 1, [1564].log_data[19].valid := 1,
        [1564].time.Year := 2023, [1564].time.Month := 1, [1564].time.Day := 15, [1564].time.Hour := 2, [1564].time.Minute := 44, [1564].time.Second := 59, [1565].log_data[0].min := 1.0, [1565].log_data[0].max := 1.0, [1565].log_data[0].total := 300.0, [1565].log_data[0].time := 300.0, [1565].log_data[0].minminute := 45, [1565].log_data[0].maxminute := 45, [1565].log_data[0].valid := 1, [1565].log_data[1].valid := 1, [1565].log_data[2].valid := 1, [1565].log_data[3].valid := 1, [1565].log_data[4].valid := 1, [1565].log_data[5].valid := 1, [1565].log_data[6].valid := 1, [1565].log_data[7].valid := 1, [1565].log_data[8].valid := 1, [1565].log_data[9].valid := 1, [1565].log_data[10].valid := 1, [1565].log_data[11].valid := 1, [1565].log_data[12].valid := 1, [1565].log_data[13].valid := 1, [1565].log_data[14].valid := 1, [1565].log_data[15].valid := 1, [1565].log_data[16].valid := 1, [1565].log_data[17].valid := 1, [1565].log_data[18].valid := 1, [1565].log_data[19].valid := 1, [1565].time.Year := 2023, [1565].time.Month := 1, [1565].time.Day := 15, [1565].time.Hour := 2, [1565].time.Minute := 49, [1565].time.Second := 59, [1566].log_data[0].min := 1.0, [1566].log_data[0].max := 1.0, [1566].log_data[0].total := 300.0, [1566].log_data[0].time := 300.0, [1566].log_data[0].minminute := 50, [1566].log_data[0].maxminute := 50, [1566].log_data[0].valid := 1, [1566].log_data[1].valid := 1, [1566].log_data[2].valid := 1, [1566].log_data[3].valid := 1, [1566].log_data[4].valid := 1, [1566].log_data[5].valid := 1, [1566].log_data[6].valid := 1, [1566].log_data[7].valid := 1, [1566].log_data[8].valid := 1, [1566].log_data[9].valid := 1, [1566].log_data[10].valid := 1, [1566].log_data[11].valid := 1, [1566].log_data[12].valid := 1, [1566].log_data[13].valid := 1, [1566].log_data[14].valid := 1, [1566].log_data[15].valid := 1,
        [1566].log_data[16].valid := 1, [1566].log_data[17].valid := 1, [1566].log_data[18].valid := 1, [1566].log_data[19].valid := 1, [1566].time.Year := 2023, [1566].time.Month := 1, [1566].time.Day := 15, [1566].time.Hour := 2, [1566].time.Minute := 54, [1566].time.Second := 59, [1567].log_data[0].min := 1.0, [1567].log_data[0].max := 1.0, [1567].log_data[0].total := 300.0, [1567].log_data[0].time := 300.0, [1567].log_data[0].minminute := 55, [1567].log_data[0].maxminute := 55, [1567].log_data[0].valid := 1, [1567].log_data[1].valid := 1, [1567].log_data[2].valid := 1, [1567].log_data[3].valid := 1, [1567].log_data[4].valid := 1, [1567].log_data[5].valid := 1, [1567].log_data[6].valid := 1, [1567].log_data[7].valid := 1, [1567].log_data[8].valid := 1, [1567].log_data[9].valid := 1, [1567].log_data[10].valid := 1, [1567].log_data[11].valid := 1, [1567].log_data[12].valid := 1, [1567].log_data[13].valid := 1, [1567].log_data[14].valid := 1, [1567].log_data[15].valid := 1, [1567].log_data[16].valid := 1, [1567].log_data[17].valid := 1, [1567].log_data[18].valid := 1, [1567].log_data[19].valid := 1, [1567].time.Year := 2023, [1567].time.Month := 1, [1567].time.Day := 15, [1567].time.Hour := 2, [1567].time.Minute := 59, [1567].time.Second := 59, [1568].log_data[0].min := 1.0, [1568].log_data[0].max := 1.0, [1568].log_data[0].total := 300.0, [1568].log_data[0].time := 300.0, [1568].log_data[0].valid := 1, [1568].log_data[1].valid := 1, [1568].log_data[2].valid := 1, [1568].log_data[3].valid := 1, [1568].log_data[4].valid := 1, [1568].log_data[5].valid := 1, [1568].log_data[6].valid := 1, [1568].log_data[7].valid := 1, [1568].log_data[8].valid := 1, [1568].log_data[9].valid := 1, [1568].log_data[10].valid := 1, [1568].log_data[11].valid := 1, [1568].log_data[12].valid := 1, [1568].log_data[13].valid := 1,
        [1568].log_data[14].valid := 1, [1568].log_data[15].valid := 1, [1568].log_data[16].valid := 1, [1568].log_data[17].valid := 1, [1568].log_data[18].valid := 1, [1568].log_data[19].valid := 1, [1568].time.Year := 2023, [1568].time.Month := 1, [1568].time.Day := 15, [1568].time.Hour := 3, [1568].time.Minute := 4, [1568].time.Second := 59, [1569].log_data[0].min := 1.0, [1569].log_data[0].max := 1.0, [1569].log_data[0].total := 300.0, [1569].log_data[0].time := 300.0, [1569].log_data[0].minminute := 5, [1569].log_data[0].maxminute := 5, [1569].log_data[0].valid := 1, [1569].log_data[1].valid := 1, [1569].log_data[2].valid := 1, [1569].log_data[3].valid := 1, [1569].log_data[4].valid := 1, [1569].log_data[5].valid := 1, [1569].log_data[6].valid := 1, [1569].log_data[7].valid := 1, [1569].log_data[8].valid := 1, [1569].log_data[9].valid := 1, [1569].log_data[10].valid := 1, [1569].log_data[11].valid := 1, [1569].log_data[12].valid := 1, [1569].log_data[13].valid := 1, [1569].log_data[14].valid := 1, [1569].log_data[15].valid := 1, [1569].log_data[16].valid := 1, [1569].log_data[17].valid := 1, [1569].log_data[18].valid := 1, [1569].log_data[19].valid := 1, [1569].time.Year := 2023, [1569].time.Month := 1, [1569].time.Day := 15, [1569].time.Hour := 3, [1569].time.Minute := 9, [1569].time.Second := 59, [1570].log_data[0].min := 1.0, [1570].log_data[0].max := 1.0, [1570].log_data[0].total := 300.0, [1570].log_data[0].time := 300.0, [1570].log_data[0].minminute := 10, [1570].log_data[0].maxminute := 10, [1570].log_data[0].valid := 1, [1570].log_data[1].valid := 1, [1570].log_data[2].valid := 1, [1570].log_data[3].valid := 1, [1570].log_data[4].valid := 1, [1570].log_data[5].valid := 1, [1570].log_data[6].valid := 1, [1570].log_data[7].valid := 1, [1570].log_data[8].valid := 1, [1570].log_data[9].valid := 1,
        [1570].log_data[10].valid := 1, [1570].log_data[11].valid := 1, [1570].log_data[12].valid := 1, [1570].log_data[13].valid := 1, [1570].log_data[14].valid := 1, [1570].log_data[15].valid := 1, [1570].log_data[16].valid := 1, [1570].log_data[17].valid := 1, [1570].log_data[18].valid := 1, [1570].log_data[19].valid := 1, [1570].time.Year := 2023, [1570].time.Month := 1, [1570].time.Day := 15, [1570].time.Hour := 3, [1570].time.Minute := 14, [1570].time.Second := 59, [1571].log_data[0].min := 1.0, [1571].log_data[0].max := 1.0, [1571].log_data[0].total := 300.0, [1571].log_data[0].time := 300.0, [1571].log_data[0].minminute := 15, [1571].log_data[0].maxminute := 15, [1571].log_data[0].valid := 1, [1571].log_data[1].valid := 1, [1571].log_data[2].valid := 1, [1571].log_data[3].valid := 1, [1571].log_data[4].valid := 1, [1571].log_data[5].valid := 1, [1571].log_data[6].valid := 1, [1571].log_data[7].valid := 1, [1571].log_data[8].valid := 1, [1571].log_data[9].valid := 1, [1571].log_data[10].valid := 1, [1571].log_data[11].valid := 1, [1571].log_data[12].valid := 1, [1571].log_data[13].valid := 1, [1571].log_data[14].valid := 1, [1571].log_data[15].valid := 1, [1571].log_data[16].valid := 1, [1571].log_data[17].valid := 1, [1571].log_data[18].valid := 1, [1571].log_data[19].valid := 1, [1571].time.Year := 2023, [1571].time.Month := 1, [1571].time.Day := 15, [1571].time.Hour := 3, [1571].time.Minute := 19, [1571].time.Second := 59, [1572].log_data[0].min := 1.0, [1572].log_data[0].max := 1.0, [1572].log_data[0].total := 300.0, [1572].log_data[0].time := 300.0, [1572].log_data[0].minminute := 20, [1572].log_data[0].maxminute := 20, [1572].log_data[0].valid := 1, [1572].log_data[1].valid := 1, [1572].log_data[2].valid := 1, [1572].log_data[3].valid := 1, [1572].log_data[4].valid := 1, [1572].log_data[5].valid := 1,
        [1572].log_data[6].valid := 1, [1572].log_data[7].valid := 1, [1572].log_data[8].valid := 1, [1572].log_data[9].valid := 1, [1572].log_data[10].valid := 1, [1572].log_data[11].valid := 1, [1572].log_data[12].valid := 1, [1572].log_data[13].valid := 1, [1572].log_data[14].valid := 1, [1572].log_data[15].valid := 1, [1572].log_data[16].valid := 1, [1572].log_data[17].valid := 1, [1572].log_data[18].valid := 1, [1572].log_data[19].valid := 1, [1572].time.Year := 2023, [1572].time.Month := 1, [1572].time.Day := 15, [1572].time.Hour := 3, [1572].time.Minute := 24, [1572].time.Second := 59, [1573].log_data[0].min := 1.0, [1573].log_data[0].max := 1.0, [1573].log_data[0].total := 300.0, [1573].log_data[0].time := 300.0, [1573].log_data[0].minminute := 25, [1573].log_data[0].maxminute := 25, [1573].log_data[0].valid := 1, [1573].log_data[1].valid := 1, [1573].log_data[2].valid := 1, [1573].log_data[3].valid := 1, [1573].log_data[4].valid := 1, [1573].log_data[5].valid := 1, [1573].log_data[6].valid := 1, [1573].log_data[7].valid := 1, [1573].log_data[8].valid := 1, [1573].log_data[9].valid := 1, [1573].log_data[10].valid := 1, [1573].log_data[11].valid := 1, [1573].log_data[12].valid := 1, [1573].log_data[13].valid := 1, [1573].log_data[14].valid := 1, [1573].log_data[15].valid := 1, [1573].log_data[16].valid := 1, [1573].log_data[17].valid := 1, [1573].log_data[18].valid := 1, [1573].log_data[19].valid := 1, [1573].time.Year := 2023, [1573].time.Month := 1, [1573].time.Day := 15, [1573].time.Hour := 3, [1573].time.Minute := 29, [1573].time.Second := 59, [1574].log_data[0].min := 1.0, [1574].log_data[0].max := 1.0, [1574].log_data[0].total := 300.0, [1574].log_data[0].time := 300.0, [1574].log_data[0].minminute := 30, [1574].log_data[0].maxminute := 30, [1574].log_data[0].valid := 1, [1574].log_data[1].valid := 1,
        [1574].log_data[2].valid := 1, [1574].log_data[3].valid := 1, [1574].log_data[4].valid := 1, [1574].log_data[5].valid := 1, [1574].log_data[6].valid := 1, [1574].log_data[7].valid := 1, [1574].log_data[8].valid := 1, [1574].log_data[9].valid := 1, [1574].log_data[10].valid := 1, [1574].log_data[11].valid := 1, [1574].log_data[12].valid := 1, [1574].log_data[13].valid := 1, [1574].log_data[14].valid := 1, [1574].log_data[15].valid := 1, [1574].log_data[16].valid := 1, [1574].log_data[17].valid := 1, [1574].log_data[18].valid := 1, [1574].log_data[19].valid := 1, [1574].time.Year := 2023, [1574].time.Month := 1, [1574].time.Day := 15, [1574].time.Hour := 3, [1574].time.Minute := 34, [1574].time.Second := 59, [1575].log_data[0].min := 1.0, [1575].log_data[0].max := 1.0, [1575].log_data[0].total := 300.0, [1575].log_data[0].time := 300.0, [1575].log_data[0].minminute := 35, [1575].log_data[0].maxminute := 35, [1575].log_data[0].valid := 1, [1575].log_data[1].valid := 1, [1575].log_data[2].valid := 1, [1575].log_data[3].valid := 1, [1575].log_data[4].valid := 1, [1575].log_data[5].valid := 1, [1575].log_data[6].valid := 1, [1575].log_data[7].valid := 1, [1575].log_data[8].valid := 1, [1575].log_data[9].valid := 1, [1575].log_data[10].valid := 1, [1575].log_data[11].valid := 1, [1575].log_data[12].valid := 1, [1575].log_data[13].valid := 1, [1575].log_data[14].valid := 1, [1575].log_data[15].valid := 1, [1575].log_data[16].valid := 1, [1575].log_data[17].valid := 1, [1575].log_data[18].valid := 1, [1575].log_data[19].valid := 1, [1575].time.Year := 2023, [1575].time.Month := 1, [1575].time.Day := 15, [1575].time.Hour := 3, [1575].time.Minute := 39, [1575].time.Second := 59, [1576].log_data[0].min := 1.0, [1576].log_data[0].max := 1.0, [1576].log_data[0].total := 300.0, [1576].log_data[0].time := 300.0,
        [1576].log_data[0].minminute := 40, [1576].log_data[0].maxminute := 40, [1576].log_data[0].valid := 1, [1576].log_data[1].valid := 1, [1576].log_data[2].valid := 1, [1576].log_data[3].valid := 1, [1576].log_data[4].valid := 1, [1576].log_data[5].valid := 1, [1576].log_data[6].valid := 1, [1576].log_data[7].valid := 1, [1576].log_data[8].valid := 1, [1576].log_data[9].valid := 1, [1576].log_data[10].valid := 1, [1576].log_data[11].valid := 1, [1576].log_data[12].valid := 1, [1576].log_data[13].valid := 1, [1576].log_data[14].valid := 1, [1576].log_data[15].valid := 1, [1576].log_data[16].valid := 1, [1576].log_data[17].valid := 1, [1576].log_data[18].valid := 1, [1576].log_data[19].valid := 1, [1576].time.Year := 2023, [1576].time.Month := 1, [1576].time.Day := 15, [1576].time.Hour := 3, [1576].time.Minute := 44, [1576].time.Second := 59, [1577].log_data[0].min := 1.0, [1577].log_data[0].max := 1.0, [1577].log_data[0].total := 300.0, [1577].log_data[0].time := 300.0, [1577].log_data[0].minminute := 45, [1577].log_data[0].maxminute := 45, [1577].log_data[0].valid := 1, [1577].log_data[1].valid := 1, [1577].log_data[2].valid := 1, [1577].log_data[3].valid := 1, [1577].log_data[4].valid := 1, [1577].log_data[5].valid := 1, [1577].log_data[6].valid := 1, [1577].log_data[7].valid := 1, [1577].log_data[8].valid := 1, [1577].log_data[9].valid := 1, [1577].log_data[10].valid := 1, [1577].log_data[11].valid := 1, [1577].log_data[12].valid := 1, [1577].log_data[13].valid := 1, [1577].log_data[14].valid := 1, [1577].log_data[15].valid := 1, [1577].log_data[16].valid := 1, [1577].log_data[17].valid := 1, [1577].log_data[18].valid := 1, [1577].log_data[19].valid := 1, [1577].time.Year := 2023, [1577].time.Month := 1, [1577].time.Day := 15, [1577].time.Hour := 3, [1577].time.Minute := 49, [1577].time.Second := 59,
        [1578].log_data[0].min := 1.0, [1578].log_data[0].max := 1.0, [1578].log_data[0].total := 300.0, [1578].log_data[0].time := 300.0, [1578].log_data[0].minminute := 50, [1578].log_data[0].maxminute := 50, [1578].log_data[0].valid := 1, [1578].log_data[1].valid := 1, [1578].log_data[2].valid := 1, [1578].log_data[3].valid := 1, [1578].log_data[4].valid := 1, [1578].log_data[5].valid := 1, [1578].log_data[6].valid := 1, [1578].log_data[7].valid := 1, [1578].log_data[8].valid := 1, [1578].log_data[9].valid := 1, [1578].log_data[10].valid := 1, [1578].log_data[11].valid := 1, [1578].log_data[12].valid := 1, [1578].log_data[13].valid := 1, [1578].log_data[14].valid := 1, [1578].log_data[15].valid := 1, [1578].log_data[16].valid := 1, [1578].log_data[17].valid := 1, [1578].log_data[18].valid := 1, [1578].log_data[19].valid := 1, [1578].time.Year := 2023, [1578].time.Month := 1, [1578].time.Day := 15, [1578].time.Hour := 3, [1578].time.Minute := 54, [1578].time.Second := 59, [1579].log_data[0].min := 1.0, [1579].log_data[0].max := 1.0, [1579].log_data[0].total := 300.0, [1579].log_data[0].time := 300.0, [1579].log_data[0].minminute := 55, [1579].log_data[0].maxminute := 55, [1579].log_data[0].valid := 1, [1579].log_data[1].valid := 1, [1579].log_data[2].valid := 1, [1579].log_data[3].valid := 1, [1579].log_data[4].valid := 1, [1579].log_data[5].valid := 1, [1579].log_data[6].valid := 1, [1579].log_data[7].valid := 1, [1579].log_data[8].valid := 1, [1579].log_data[9].valid := 1, [1579].log_data[10].valid := 1, [1579].log_data[11].valid := 1, [1579].log_data[12].valid := 1, [1579].log_data[13].valid := 1, [1579].log_data[14].valid := 1, [1579].log_data[15].valid := 1, [1579].log_data[16].valid := 1, [1579].log_data[17].valid := 1, [1579].log_data[18].valid := 1, [1579].log_data[19].valid := 1, [1579].time.Year := 2023, [1579].time.Month := 1,
        [1579].time.Day := 15, [1579].time.Hour := 3, [1579].time.Minute := 59, [1579].time.Second := 59, [1580].log_data[0].min := 1.0, [1580].log_data[0].max := 1.0, [1580].log_data[0].total := 300.0, [1580].log_data[0].time := 300.0, [1580].log_data[0].valid := 1, [1580].log_data[1].valid := 1, [1580].log_data[2].valid := 1, [1580].log_data[3].valid := 1, [1580].log_data[4].valid := 1, [1580].log_data[5].valid := 1, [1580].log_data[6].valid := 1, [1580].log_data[7].valid := 1, [1580].log_data[8].valid := 1, [1580].log_data[9].valid := 1, [1580].log_data[10].valid := 1, [1580].log_data[11].valid := 1, [1580].log_data[12].valid := 1, [1580].log_data[13].valid := 1, [1580].log_data[14].valid := 1, [1580].log_data[15].valid := 1, [1580].log_data[16].valid := 1, [1580].log_data[17].valid := 1, [1580].log_data[18].valid := 1, [1580].log_data[19].valid := 1, [1580].time.Year := 2023, [1580].time.Month := 1, [1580].time.Day := 15, [1580].time.Hour := 4, [1580].time.Minute := 4, [1580].time.Second := 59, [1581].log_data[0].min := 1.0, [1581].log_data[0].max := 1.0, [1581].log_data[0].total := 300.0, [1581].log_data[0].time := 300.0, [1581].log_data[0].minminute := 5, [1581].log_data[0].maxminute := 5, [1581].log_data[0].valid := 1, [1581].log_data[1].valid := 1, [1581].log_data[2].valid := 1, [1581].log_data[3].valid := 1, [1581].log_data[4].valid := 1, [1581].log_data[5].valid := 1, [1581].log_data[6].valid := 1, [1581].log_data[7].valid := 1, [1581].log_data[8].valid := 1, [1581].log_data[9].valid := 1, [1581].log_data[10].valid := 1, [1581].log_data[11].valid := 1, [1581].log_data[12].valid := 1, [1581].log_data[13].valid := 1, [1581].log_data[14].valid := 1, [1581].log_data[15].valid := 1, [1581].log_data[16].valid := 1, [1581].log_data[17].valid := 1, [1581].log_data[18].valid := 1, [1581].log_data[19].valid := 1,
        [1581].time.Year := 2023, [1581].time.Month := 1, [1581].time.Day := 15, [1581].time.Hour := 4, [1581].time.Minute := 9, [1581].time.Second := 59, [1582].log_data[0].min := 1.0, [1582].log_data[0].max := 1.0, [1582].log_data[0].total := 300.0, [1582].log_data[0].time := 300.0, [1582].log_data[0].minminute := 10, [1582].log_data[0].maxminute := 10, [1582].log_data[0].valid := 1, [1582].log_data[1].valid := 1, [1582].log_data[2].valid := 1, [1582].log_data[3].valid := 1, [1582].log_data[4].valid := 1, [1582].log_data[5].valid := 1, [1582].log_data[6].valid := 1, [1582].log_data[7].valid := 1, [1582].log_data[8].valid := 1, [1582].log_data[9].valid := 1, [1582].log_data[10].valid := 1, [1582].log_data[11].valid := 1, [1582].log_data[12].valid := 1, [1582].log_data[13].valid := 1, [1582].log_data[14].valid := 1, [1582].log_data[15].valid := 1, [1582].log_data[16].valid := 1, [1582].log_data[17].valid := 1, [1582].log_data[18].valid := 1, [1582].log_data[19].valid := 1, [1582].time.Year := 2023, [1582].time.Month := 1, [1582].time.Day := 15, [1582].time.Hour := 4, [1582].time.Minute := 14, [1582].time.Second := 59, [1583].log_data[0].min := 1.0, [1583].log_data[0].max := 1.0, [1583].log_data[0].total := 300.0, [1583].log_data[0].time := 300.0, [1583].log_data[0].minminute := 15, [1583].log_data[0].maxminute := 15, [1583].log_data[0].valid := 1, [1583].log_data[1].valid := 1, [1583].log_data[2].valid := 1, [1583].log_data[3].valid := 1, [1583].log_data[4].valid := 1, [1583].log_data[5].valid := 1, [1583].log_data[6].valid := 1, [1583].log_data[7].valid := 1, [1583].log_data[8].valid := 1, [1583].log_data[9].valid := 1, [1583].log_data[10].valid := 1, [1583].log_data[11].valid := 1, [1583].log_data[12].valid := 1, [1583].log_data[13].valid := 1, [1583].log_data[14].valid := 1, [1583].log_data[15].valid := 1,
        [1583].log_data[16].valid := 1, [1583].log_data[17].valid := 1, [1583].log_data[18].valid := 1, [1583].log_data[19].valid := 1, [1583].time.Year := 2023, [1583].time.Month := 1, [1583].time.Day := 15, [1583].time.Hour := 4, [1583].time.Minute := 19, [1583].time.Second := 59, [1584].log_data[0].min := 1.0, [1584].log_data[0].max := 1.0, [1584].log_data[0].total := 300.0, [1584].log_data[0].time := 300.0, [1584].log_data[0].minminute := 20, [1584].log_data[0].maxminute := 20, [1584].log_data[0].valid := 1, [1584].log_data[1].valid := 1, [1584].log_data[2].valid := 1, [1584].log_data[3].valid := 1, [1584].log_data[4].valid := 1, [1584].log_data[5].valid := 1, [1584].log_data[6].valid := 1, [1584].log_data[7].valid := 1, [1584].log_data[8].valid := 1, [1584].log_data[9].valid := 1, [1584].log_data[10].valid := 1, [1584].log_data[11].valid := 1, [1584].log_data[12].valid := 1, [1584].log_data[13].valid := 1, [1584].log_data[14].valid := 1, [1584].log_data[15].valid := 1, [1584].log_data[16].valid := 1, [1584].log_data[17].valid := 1, [1584].log_data[18].valid := 1, [1584].log_data[19].valid := 1, [1584].time.Year := 2023, [1584].time.Month := 1, [1584].time.Day := 15, [1584].time.Hour := 4, [1584].time.Minute := 24, [1584].time.Second := 59, [1585].log_data[0].min := 1.0, [1585].log_data[0].max := 1.0, [1585].log_data[0].total := 300.0, [1585].log_data[0].time := 300.0, [1585].log_data[0].minminute := 25, [1585].log_data[0].maxminute := 25, [1585].log_data[0].valid := 1, [1585].log_data[1].valid := 1, [1585].log_data[2].valid := 1, [1585].log_data[3].valid := 1, [1585].log_data[4].valid := 1, [1585].log_data[5].valid := 1, [1585].log_data[6].valid := 1, [1585].log_data[7].valid := 1, [1585].log_data[8].valid := 1, [1585].log_data[9].valid := 1, [1585].log_data[10].valid := 1, [1585].log_data[11].valid := 1,
        [1585].log_data[12].valid := 1, [1585].log_data[13].valid := 1, [1585].log_data[14].valid := 1, [1585].log_data[15].valid := 1, [1585].log_data[16].valid := 1, [1585].log_data[17].valid := 1, [1585].log_data[18].valid := 1, [1585].log_data[19].valid := 1, [1585].time.Year := 2023, [1585].time.Month := 1, [1585].time.Day := 15, [1585].time.Hour := 4, [1585].time.Minute := 29, [1585].time.Second := 59, [1586].log_data[0].min := 1.0, [1586].log_data[0].max := 1.0, [1586].log_data[0].total := 300.0, [1586].log_data[0].time := 300.0, [1586].log_data[0].minminute := 30, [1586].log_data[0].maxminute := 30, [1586].log_data[0].valid := 1, [1586].log_data[1].valid := 1, [1586].log_data[2].valid := 1, [1586].log_data[3].valid := 1, [1586].log_data[4].valid := 1, [1586].log_data[5].valid := 1, [1586].log_data[6].valid := 1, [1586].log_data[7].valid := 1, [1586].log_data[8].valid := 1, [1586].log_data[9].valid := 1, [1586].log_data[10].valid := 1, [1586].log_data[11].valid := 1, [1586].log_data[12].valid := 1, [1586].log_data[13].valid := 1, [1586].log_data[14].valid := 1, [1586].log_data[15].valid := 1, [1586].log_data[16].valid := 1, [1586].log_data[17].valid := 1, [1586].log_data[18].valid := 1, [1586].log_data[19].valid := 1, [1586].time.Year := 2023, [1586].time.Month := 1, [1586].time.Day := 15, [1586].time.Hour := 4, [1586].time.Minute := 34, [1586].time.Second := 59, [1587].log_data[0].min := 1.0, [1587].log_data[0].max := 1.0, [1587].log_data[0].total := 300.0, [1587].log_data[0].time := 300.0, [1587].log_data[0].minminute := 35, [1587].log_data[0].maxminute := 35, [1587].log_data[0].valid := 1, [1587].log_data[1].valid := 1, [1587].log_data[2].valid := 1, [1587].log_data[3].valid := 1, [1587].log_data[4].valid := 1, [1587].log_data[5].valid := 1, [1587].log_data[6].valid := 1, [1587].log_data[7].valid := 1,
        [1587].log_data[8].valid := 1, [1587].log_data[9].valid := 1, [1587].log_data[10].valid := 1, [1587].log_data[11].valid := 1, [1587].log_data[12].valid := 1, [1587].log_data[13].valid := 1, [1587].log_data[14].valid := 1, [1587].log_data[15].valid := 1, [1587].log_data[16].valid := 1, [1587].log_data[17].valid := 1, [1587].log_data[18].valid := 1, [1587].log_data[19].valid := 1, [1587].time.Year := 2023, [1587].time.Month := 1, [1587].time.Day := 15, [1587].time.Hour := 4, [1587].time.Minute := 39, [1587].time.Second := 59, [1588].log_data[0].min := 1.0, [1588].log_data[0].max := 1.0, [1588].log_data[0].total := 300.0, [1588].log_data[0].time := 300.0, [1588].log_data[0].minminute := 40, [1588].log_data[0].maxminute := 40, [1588].log_data[0].valid := 1, [1588].log_data[1].valid := 1, [1588].log_data[2].valid := 1, [1588].log_data[3].valid := 1, [1588].log_data[4].valid := 1, [1588].log_data[5].valid := 1, [1588].log_data[6].valid := 1, [1588].log_data[7].valid := 1, [1588].log_data[8].valid := 1, [1588].log_data[9].valid := 1, [1588].log_data[10].valid := 1, [1588].log_data[11].valid := 1, [1588].log_data[12].valid := 1, [1588].log_data[13].valid := 1, [1588].log_data[14].valid := 1, [1588].log_data[15].valid := 1, [1588].log_data[16].valid := 1, [1588].log_data[17].valid := 1, [1588].log_data[18].valid := 1, [1588].log_data[19].valid := 1, [1588].time.Year := 2023, [1588].time.Month := 1, [1588].time.Day := 15, [1588].time.Hour := 4, [1588].time.Minute := 44, [1588].time.Second := 59, [1589].log_data[0].min := 1.0, [1589].log_data[0].max := 1.0, [1589].log_data[0].total := 300.0, [1589].log_data[0].time := 300.0, [1589].log_data[0].minminute := 45, [1589].log_data[0].maxminute := 45, [1589].log_data[0].valid := 1, [1589].log_data[1].valid := 1, [1589].log_data[2].valid := 1, [1589].log_data[3].valid := 1,
        [1589].log_data[4].valid := 1, [1589].log_data[5].valid := 1, [1589].log_data[6].valid := 1, [1589].log_data[7].valid := 1, [1589].log_data[8].valid := 1, [1589].log_data[9].valid := 1, [1589].log_data[10].valid := 1, [1589].log_data[11].valid := 1, [1589].log_data[12].valid := 1, [1589].log_data[13].valid := 1, [1589].log_data[14].valid := 1, [1589].log_data[15].valid := 1, [1589].log_data[16].valid := 1, [1589].log_data[17].valid := 1, [1589].log_data[18].valid := 1, [1589].log_data[19].valid := 1, [1589].time.Year := 2023, [1589].time.Month := 1, [1589].time.Day := 15, [1589].time.Hour := 4, [1589].time.Minute := 49, [1589].time.Second := 59, [1590].log_data[0].min := 1.0, [1590].log_data[0].max := 1.0, [1590].log_data[0].total := 300.0, [1590].log_data[0].time := 300.0, [1590].log_data[0].minminute := 50, [1590].log_data[0].maxminute := 50, [1590].log_data[0].valid := 1, [1590].log_data[1].valid := 1, [1590].log_data[2].valid := 1, [1590].log_data[3].valid := 1, [1590].log_data[4].valid := 1, [1590].log_data[5].valid := 1, [1590].log_data[6].valid := 1, [1590].log_data[7].valid := 1, [1590].log_data[8].valid := 1, [1590].log_data[9].valid := 1, [1590].log_data[10].valid := 1, [1590].log_data[11].valid := 1, [1590].log_data[12].valid := 1, [1590].log_data[13].valid := 1, [1590].log_data[14].valid := 1, [1590].log_data[15].valid := 1, [1590].log_data[16].valid := 1, [1590].log_data[17].valid := 1, [1590].log_data[18].valid := 1, [1590].log_data[19].valid := 1, [1590].time.Year := 2023, [1590].time.Month := 1, [1590].time.Day := 15, [1590].time.Hour := 4, [1590].time.Minute := 54, [1590].time.Second := 59, [1591].log_data[0].min := 1.0, [1591].log_data[0].max := 1.0, [1591].log_data[0].total := 300.0, [1591].log_data[0].time := 300.0, [1591].log_data[0].minminute := 55, [1591].log_data[0].maxminute := 55,
        [1591].log_data[0].valid := 1, [1591].log_data[1].valid := 1, [1591].log_data[2].valid := 1, [1591].log_data[3].valid := 1, [1591].log_data[4].valid := 1, [1591].log_data[5].valid := 1, [1591].log_data[6].valid := 1, [1591].log_data[7].valid := 1, [1591].log_data[8].valid := 1, [1591].log_data[9].valid := 1, [1591].log_data[10].valid := 1, [1591].log_data[11].valid := 1, [1591].log_data[12].valid := 1, [1591].log_data[13].valid := 1, [1591].log_data[14].valid := 1, [1591].log_data[15].valid := 1, [1591].log_data[16].valid := 1, [1591].log_data[17].valid := 1, [1591].log_data[18].valid := 1, [1591].log_data[19].valid := 1, [1591].time.Year := 2023, [1591].time.Month := 1, [1591].time.Day := 15, [1591].time.Hour := 4, [1591].time.Minute := 59, [1591].time.Second := 59, [1592].log_data[0].min := 1.0, [1592].log_data[0].max := 1.0, [1592].log_data[0].total := 300.0, [1592].log_data[0].time := 300.0, [1592].log_data[0].valid := 1, [1592].log_data[1].valid := 1, [1592].log_data[2].valid := 1, [1592].log_data[3].valid := 1, [1592].log_data[4].valid := 1, [1592].log_data[5].valid := 1, [1592].log_data[6].valid := 1, [1592].log_data[7].valid := 1, [1592].log_data[8].valid := 1, [1592].log_data[9].valid := 1, [1592].log_data[10].valid := 1, [1592].log_data[11].valid := 1, [1592].log_data[12].valid := 1, [1592].log_data[13].valid := 1, [1592].log_data[14].valid := 1, [1592].log_data[15].valid := 1, [1592].log_data[16].valid := 1, [1592].log_data[17].valid := 1, [1592].log_data[18].valid := 1, [1592].log_data[19].valid := 1, [1592].time.Year := 2023, [1592].time.Month := 1, [1592].time.Day := 15, [1592].time.Hour := 5, [1592].time.Minute := 4, [1592].time.Second := 59, [1593].log_data[0].min := 1.0, [1593].log_data[0].max := 1.0, [1593].log_data[0].total := 300.0, [1593].log_data[0].time := 300.0,
        [1593].log_data[0].minminute := 5, [1593].log_data[0].maxminute := 5, [1593].log_data[0].valid := 1, [1593].log_data[1].valid := 1, [1593].log_data[2].valid := 1, [1593].log_data[3].valid := 1, [1593].log_data[4].valid := 1, [1593].log_data[5].valid := 1, [1593].log_data[6].valid := 1, [1593].log_data[7].valid := 1, [1593].log_data[8].valid := 1, [1593].log_data[9].valid := 1, [1593].log_data[10].valid := 1, [1593].log_data[11].valid := 1, [1593].log_data[12].valid := 1, [1593].log_data[13].valid := 1, [1593].log_data[14].valid := 1, [1593].log_data[15].valid := 1, [1593].log_data[16].valid := 1, [1593].log_data[17].valid := 1, [1593].log_data[18].valid := 1, [1593].log_data[19].valid := 1, [1593].time.Year := 2023, [1593].time.Month := 1, [1593].time.Day := 15, [1593].time.Hour := 5, [1593].time.Minute := 9, [1593].time.Second := 59, [1594].log_data[0].min := 1.0, [1594].log_data[0].max := 1.0, [1594].log_data[0].total := 300.0, [1594].log_data[0].time := 300.0, [1594].log_data[0].minminute := 10, [1594].log_data[0].maxminute := 10, [1594].log_data[0].valid := 1, [1594].log_data[1].valid := 1, [1594].log_data[2].valid := 1, [1594].log_data[3].valid := 1, [1594].log_data[4].valid := 1, [1594].log_data[5].valid := 1, [1594].log_data[6].valid := 1, [1594].log_data[7].valid := 1, [1594].log_data[8].valid := 1, [1594].log_data[9].valid := 1, [1594].log_data[10].valid := 1, [1594].log_data[11].valid := 1, [1594].log_data[12].valid := 1, [1594].log_data[13].valid := 1, [1594].log_data[14].valid := 1, [1594].log_data[15].valid := 1, [1594].log_data[16].valid := 1, [1594].log_data[17].valid := 1, [1594].log_data[18].valid := 1, [1594].log_data[19].valid := 1, [1594].time.Year := 2023, [1594].time.Month := 1, [1594].time.Day := 15, [1594].time.Hour := 5, [1594].time.Minute := 14, [1594].time.Second := 59,
        [1595].log_data[0].min := 1.0, [1595].log_data[0].max := 1.0, [1595].log_data[0].total := 300.0, [1595].log_data[0].time := 300.0, [1595].log_data[0].minminute := 15, [1595].log_data[0].maxminute := 15, [1595].log_data[0].valid := 1, [1595].log_data[1].valid := 1, [1595].log_data[2].valid := 1, [1595].log_data[3].valid := 1, [1595].log_data[4].valid := 1, [1595].log_data[5].valid := 1, [1595].log_data[6].valid := 1, [1595].log_data[7].valid := 1, [1595].log_data[8].valid := 1, [1595].log_data[9].valid := 1, [1595].log_data[10].valid := 1, [1595].log_data[11].valid := 1, [1595].log_data[12].valid := 1, [1595].log_data[13].valid := 1, [1595].log_data[14].valid := 1, [1595].log_data[15].valid := 1, [1595].log_data[16].valid := 1, [1595].log_data[17].valid := 1, [1595].log_data[18].valid := 1, [1595].log_data[19].valid := 1, [1595].time.Year := 2023, [1595].time.Month := 1, [1595].time.Day := 15, [1595].time.Hour := 5, [1595].time.Minute := 19, [1595].time.Second := 59, [1596].log_data[0].min := 1.0, [1596].log_data[0].max := 1.0, [1596].log_data[0].total := 300.0, [1596].log_data[0].time := 300.0, [1596].log_data[0].minminute := 20, [1596].log_data[0].maxminute := 20, [1596].log_data[0].valid := 1, [1596].log_data[1].valid := 1, [1596].log_data[2].valid := 1, [1596].log_data[3].valid := 1, [1596].log_data[4].valid := 1, [1596].log_data[5].valid := 1, [1596].log_data[6].valid := 1, [1596].log_data[7].valid := 1, [1596].log_data[8].valid := 1, [1596].log_data[9].valid := 1, [1596].log_data[10].valid := 1, [1596].log_data[11].valid := 1, [1596].log_data[12].valid := 1, [1596].log_data[13].valid := 1, [1596].log_data[14].valid := 1, [1596].log_data[15].valid := 1, [1596].log_data[16].valid := 1, [1596].log_data[17].valid := 1, [1596].log_data[18].valid := 1, [1596].log_data[19].valid := 1, [1596].time.Year := 2023, [1596].time.Month := 1,
        [1596].time.Day := 15, [1596].time.Hour := 5, [1596].time.Minute := 24, [1596].time.Second := 59, [1597].log_data[0].min := 1.0, [1597].log_data[0].max := 1.0, [1597].log_data[0].total := 300.0, [1597].log_data[0].time := 300.0, [1597].log_data[0].minminute := 25, [1597].log_data[0].maxminute := 25, [1597].log_data[0].valid := 1, [1597].log_data[1].valid := 1, [1597].log_data[2].valid := 1, [1597].log_data[3].valid := 1, [1597].log_data[4].valid := 1, [1597].log_data[5].valid := 1, [1597].log_data[6].valid := 1, [1597].log_data[7].valid := 1, [1597].log_data[8].valid := 1, [1597].log_data[9].valid := 1, [1597].log_data[10].valid := 1, [1597].log_data[11].valid := 1, [1597].log_data[12].valid := 1, [1597].log_data[13].valid := 1, [1597].log_data[14].valid := 1, [1597].log_data[15].valid := 1, [1597].log_data[16].valid := 1, [1597].log_data[17].valid := 1, [1597].log_data[18].valid := 1, [1597].log_data[19].valid := 1, [1597].time.Year := 2023, [1597].time.Month := 1, [1597].time.Day := 15, [1597].time.Hour := 5, [1597].time.Minute := 29, [1597].time.Second := 59, [1598].log_data[0].min := 1.0, [1598].log_data[0].max := 1.0, [1598].log_data[0].total := 300.0, [1598].log_data[0].time := 300.0, [1598].log_data[0].minminute := 30, [1598].log_data[0].maxminute := 30, [1598].log_data[0].valid := 1, [1598].log_data[1].valid := 1, [1598].log_data[2].valid := 1, [1598].log_data[3].valid := 1, [1598].log_data[4].valid := 1, [1598].log_data[5].valid := 1, [1598].log_data[6].valid := 1, [1598].log_data[7].valid := 1, [1598].log_data[8].valid := 1, [1598].log_data[9].valid := 1, [1598].log_data[10].valid := 1, [1598].log_data[11].valid := 1, [1598].log_data[12].valid := 1, [1598].log_data[13].valid := 1, [1598].log_data[14].valid := 1, [1598].log_data[15].valid := 1, [1598].log_data[16].valid := 1, [1598].log_data[17].valid := 1,
        [1598].log_data[18].valid := 1, [1598].log_data[19].valid := 1, [1598].time.Year := 2023, [1598].time.Month := 1, [1598].time.Day := 15, [1598].time.Hour := 5, [1598].time.Minute := 34, [1598].time.Second := 59, [1599].log_data[0].min := 1.0, [1599].log_data[0].max := 1.0, [1599].log_data[0].total := 300.0, [1599].log_data[0].time := 300.0, [1599].log_data[0].minminute := 35, [1599].log_data[0].maxminute := 35, [1599].log_data[0].valid := 1, [1599].log_data[1].valid := 1, [1599].log_data[2].valid := 1, [1599].log_data[3].valid := 1, [1599].log_data[4].valid := 1, [1599].log_data[5].valid := 1, [1599].log_data[6].valid := 1, [1599].log_data[7].valid := 1, [1599].log_data[8].valid := 1, [1599].log_data[9].valid := 1, [1599].log_data[10].valid := 1, [1599].log_data[11].valid := 1, [1599].log_data[12].valid := 1, [1599].log_data[13].valid := 1, [1599].log_data[14].valid := 1, [1599].log_data[15].valid := 1, [1599].log_data[16].valid := 1, [1599].log_data[17].valid := 1, [1599].log_data[18].valid := 1, [1599].log_data[19].valid := 1, [1599].time.Year := 2023, [1599].time.Month := 1, [1599].time.Day := 15, [1599].time.Hour := 5, [1599].time.Minute := 39, [1599].time.Second := 59, [1600].log_data[0].min := 1.0, [1600].log_data[0].max := 1.0, [1600].log_data[0].total := 300.0, [1600].log_data[0].time := 300.0, [1600].log_data[0].minminute := 40, [1600].log_data[0].maxminute := 40, [1600].log_data[0].valid := 1, [1600].log_data[1].valid := 1, [1600].log_data[2].valid := 1, [1600].log_data[3].valid := 1, [1600].log_data[4].valid := 1, [1600].log_data[5].valid := 1, [1600].log_data[6].valid := 1, [1600].log_data[7].valid := 1, [1600].log_data[8].valid := 1, [1600].log_data[9].valid := 1, [1600].log_data[10].valid := 1, [1600].log_data[11].valid := 1, [1600].log_data[12].valid := 1, [1600].log_data[13].valid := 1,
        [1600].log_data[14].valid := 1, [1600].log_data[15].valid := 1, [1600].log_data[16].valid := 1, [1600].log_data[17].valid := 1, [1600].log_data[18].valid := 1, [1600].log_data[19].valid := 1, [1600].time.Year := 2023, [1600].time.Month := 1, [1600].time.Day := 15, [1600].time.Hour := 5, [1600].time.Minute := 44, [1600].time.Second := 59, [1601].log_data[0].min := 1.0, [1601].log_data[0].max := 1.0, [1601].log_data[0].total := 300.0, [1601].log_data[0].time := 300.0, [1601].log_data[0].minminute := 45, [1601].log_data[0].maxminute := 45, [1601].log_data[0].valid := 1, [1601].log_data[1].valid := 1, [1601].log_data[2].valid := 1, [1601].log_data[3].valid := 1, [1601].log_data[4].valid := 1, [1601].log_data[5].valid := 1, [1601].log_data[6].valid := 1, [1601].log_data[7].valid := 1, [1601].log_data[8].valid := 1, [1601].log_data[9].valid := 1, [1601].log_data[10].valid := 1, [1601].log_data[11].valid := 1, [1601].log_data[12].valid := 1, [1601].log_data[13].valid := 1, [1601].log_data[14].valid := 1, [1601].log_data[15].valid := 1, [1601].log_data[16].valid := 1, [1601].log_data[17].valid := 1, [1601].log_data[18].valid := 1, [1601].log_data[19].valid := 1, [1601].time.Year := 2023, [1601].time.Month := 1, [1601].time.Day := 15, [1601].time.Hour := 5, [1601].time.Minute := 49, [1601].time.Second := 59, [1602].log_data[0].min := 1.0, [1602].log_data[0].max := 1.0, [1602].log_data[0].total := 300.0, [1602].log_data[0].time := 300.0, [1602].log_data[0].minminute := 50, [1602].log_data[0].maxminute := 50, [1602].log_data[0].valid := 1, [1602].log_data[1].valid := 1, [1602].log_data[2].valid := 1, [1602].log_data[3].valid := 1, [1602].log_data[4].valid := 1, [1602].log_data[5].valid := 1, [1602].log_data[6].valid := 1, [1602].log_data[7].valid := 1, [1602].log_data[8].valid := 1, [1602].log_data[9].valid := 1,
        [1602].log_data[10].valid := 1, [1602].log_data[11].valid := 1, [1602].log_data[12].valid := 1, [1602].log_data[13].valid := 1, [1602].log_data[14].valid := 1, [1602].log_data[15].valid := 1, [1602].log_data[16].valid := 1, [1602].log_data[17].valid := 1, [1602].log_data[18].valid := 1, [1602].log_data[19].valid := 1, [1602].time.Year := 2023, [1602].time.Month := 1, [1602].time.Day := 15, [1602].time.Hour := 5, [1602].time.Minute := 54, [1602].time.Second := 59, [1603].log_data[0].min := 1.0, [1603].log_data[0].max := 1.0, [1603].log_data[0].total := 300.0, [1603].log_data[0].time := 300.0, [1603].log_data[0].minminute := 55, [1603].log_data[0].maxminute := 55, [1603].log_data[0].valid := 1, [1603].log_data[1].valid := 1, [1603].log_data[2].valid := 1, [1603].log_data[3].valid := 1, [1603].log_data[4].valid := 1, [1603].log_data[5].valid := 1, [1603].log_data[6].valid := 1, [1603].log_data[7].valid := 1, [1603].log_data[8].valid := 1, [1603].log_data[9].valid := 1, [1603].log_data[10].valid := 1, [1603].log_data[11].valid := 1, [1603].log_data[12].valid := 1, [1603].log_data[13].valid := 1, [1603].log_data[14].valid := 1, [1603].log_data[15].valid := 1, [1603].log_data[16].valid := 1, [1603].log_data[17].valid := 1, [1603].log_data[18].valid := 1, [1603].log_data[19].valid := 1, [1603].time.Year := 2023, [1603].time.Month := 1, [1603].time.Day := 15, [1603].time.Hour := 5, [1603].time.Minute := 59, [1603].time.Second := 59, [1604].log_data[0].min := 1.0, [1604].log_data[0].max := 1.0, [1604].log_data[0].total := 300.0, [1604].log_data[0].time := 300.0, [1604].log_data[0].valid := 1, [1604].log_data[1].valid := 1, [1604].log_data[2].valid := 1, [1604].log_data[3].valid := 1, [1604].log_data[4].valid := 1, [1604].log_data[5].valid := 1, [1604].log_data[6].valid := 1, [1604].log_data[7].valid := 1,
        [1604].log_data[8].valid := 1, [1604].log_data[9].valid := 1, [1604].log_data[10].valid := 1, [1604].log_data[11].valid := 1, [1604].log_data[12].valid := 1, [1604].log_data[13].valid := 1, [1604].log_data[14].valid := 1, [1604].log_data[15].valid := 1, [1604].log_data[16].valid := 1, [1604].log_data[17].valid := 1, [1604].log_data[18].valid := 1, [1604].log_data[19].valid := 1, [1604].time.Year := 2023, [1604].time.Month := 1, [1604].time.Day := 15, [1604].time.Hour := 6, [1604].time.Minute := 4, [1604].time.Second := 59, [1605].log_data[0].min := 1.0, [1605].log_data[0].max := 1.0, [1605].log_data[0].total := 300.0, [1605].log_data[0].time := 300.0, [1605].log_data[0].minminute := 5, [1605].log_data[0].maxminute := 5, [1605].log_data[0].valid := 1, [1605].log_data[1].valid := 1, [1605].log_data[2].valid := 1, [1605].log_data[3].valid := 1, [1605].log_data[4].valid := 1, [1605].log_data[5].valid := 1, [1605].log_data[6].valid := 1, [1605].log_data[7].valid := 1, [1605].log_data[8].valid := 1, [1605].log_data[9].valid := 1, [1605].log_data[10].valid := 1, [1605].log_data[11].valid := 1, [1605].log_data[12].valid := 1, [1605].log_data[13].valid := 1, [1605].log_data[14].valid := 1, [1605].log_data[15].valid := 1, [1605].log_data[16].valid := 1, [1605].log_data[17].valid := 1, [1605].log_data[18].valid := 1, [1605].log_data[19].valid := 1, [1605].time.Year := 2023, [1605].time.Month := 1, [1605].time.Day := 15, [1605].time.Hour := 6, [1605].time.Minute := 9, [1605].time.Second := 59, [1606].log_data[0].min := 1.0, [1606].log_data[0].max := 1.0, [1606].log_data[0].total := 300.0, [1606].log_data[0].time := 300.0, [1606].log_data[0].minminute := 10, [1606].log_data[0].maxminute := 10, [1606].log_data[0].valid := 1, [1606].log_data[1].valid := 1, [1606].log_data[2].valid := 1, [1606].log_data[3].valid := 1,
